(* IEC 61131-3 sources: SmartHomeNew/snapshots/2026-05-19, 186 files *)

(* ---- E_Adapt_Profile.dut ---- *)
{attribute 'strict'}
TYPE E_Adapt_Profile :
(
    ADAPT_PROFILE_STABLE := 0,
    ADAPT_PROFILE_BALANCED := 1,
    ADAPT_PROFILE_AGGRESSIVE := 2
) USINT;
END_TYPE

(* ---- E_FABRIC_LIFECYCLE_STATE.dut ---- *)
TYPE E_FABRIC_LIFECYCLE_STATE : (
    FABRIC_INITIALIZING,
    FABRIC_ACTIVE,
    FABRIC_DEGRADED,
    FABRIC_PASSIVE,
    FABRIC_QUARANTINED,
    FABRIC_SUSPENDED
);
END_TYPE

(* ---- E_GOVERNANCE_PRIORITY_TIER.dut ---- *)
TYPE E_GOVERNANCE_PRIORITY_TIER : (
    TIER_0_SAFETY,
    TIER_1_AUTHORITY,
    TIER_2_PHYSICAL_TRUTH,
    TIER_3_SURVIVABILITY,
    TIER_4_OBSERVABILITY,
    TIER_5_ANALYTICS
);
END_TYPE

(* ---- E_Heating_Allocation_Block_Reason.dut ---- *)
TYPE E_Heating_Allocation_Block_Reason :
(
    NONE := 0,
    PRESSURE_UNAVAILABLE := 1,
    SERVICE_DISABLED := 2,
    PREDICTIVE_DEGRADED := 3,
    POLICY_BUDGET_SHED := 4,
    FREEZE_BYPASS := 5,
    DHW_BYPASS := 6
);
END_TYPE

(* ---- E_OpenTherm_Adapter_State.dut ---- *)
TYPE E_OpenTherm_Adapter_State :
(
    OT_STATE_OFFLINE := 0,
    OT_STATE_ONLINE := 1,
    OT_STATE_HEARTBEAT_TIMEOUT := 2,
    OT_STATE_ACK_TIMEOUT := 3,
    OT_STATE_ADAPTER_ERROR := 4
);
END_TYPE

(* ---- E_PLC_ROLE.dut ---- *)
{attribute 'strict'}
TYPE E_PLC_ROLE :
(
    ROLE_UNDEFINED := 0,
    ROLE_ACTIVE := 1,
    ROLE_STANDBY := 2,
    ROLE_OFFLINE := 3
) USINT;
END_TYPE

(* ---- E_Runtime_Observer_Lifecycle_State.dut ---- *)
TYPE E_Runtime_Observer_Lifecycle_State :
(
    ROS_INACTIVE := 0,
    ROS_AUTHORIZATION_PENDING := 10,
    ROS_AUTHORIZATION_DENIED := 20,
    ROS_STABILIZATION := 30,
    ROS_OPERATIONAL := 40,
    ROS_ROLLBACK := 50,
    ROS_FAULTED := 900
);
END_TYPE

(* ---- E_SEMANTIC_EXECUTION_PATH.dut ---- *)
TYPE E_SEMANTIC_EXECUTION_PATH : (
    FAST_PATH,
    NORMAL_PATH,
    DEFERRED_PATH,
    BACKGROUND_PATH
);
END_TYPE

(* ---- E_System_Reason_Code.dut ---- *)
{attribute 'strict'}
TYPE E_System_Reason_Code :
(
    REASON_NONE := 0,
    REASON_USER := 1,
    REASON_SAFETY := 2,
    REASON_AUTOMATION := 3,
    REASON_INTERNAL := 4,
    REASON_SCENARIO_VENT_BOOST := 5,
    REASON_USER_REQUEST := 6,
    REASON_SCENARIO_NIGHT := 7,
    REASON_DOMAIN_PROJECTION := 8,
    REASON_SAFETY_BLOCK := 9
) USINT;
END_TYPE

(* ---- E_SYSTEM_RUNTIME_STATE.dut ---- *)
TYPE E_SYSTEM_RUNTIME_STATE : (
    SYS_SAFE,
    SYS_DEGRADED,
    SYS_RECOVERING,
    SYS_QUARANTINED,
    SYS_ISOLATED,
    SYS_PARTITIONED,
    SYS_TRUSTLESS
);
END_TYPE

(* ---- E_VALVE_TYPE.dut ---- *)
{attribute 'strict'}
TYPE E_VALVE_TYPE :
(
  VALVE_NC := 1,
  VALVE_NO := 2
) USINT;
END_TYPE

(* ---- E_WEATHER_COMPENSATION_METHOD.dut ---- *)
{attribute 'strict'}
TYPE E_WEATHER_COMPENSATION_METHOD :
(
  WEATHER_COMP_NONE := 0,
  WEATHER_COMP_OUTDOOR_RESET := 1
) USINT;
END_TYPE

(* ---- GVL_FABRIC_LIFECYCLE_REGISTRY.gvl ---- *)
TYPE E_FABRIC_LIFECYCLE_STATE : (
    FABRIC_INITIALIZING,
    FABRIC_ACTIVE,
    FABRIC_DEGRADED,
    FABRIC_PASSIVE,
    FABRIC_QUARANTINED,
    FABRIC_SUSPENDED
);
END_TYPE

TYPE E_RUNTIME_ADAPTIVE_MODE : (
    FULL_SEMANTIC_MODE,
    REDUCED_ANALYTICS_MODE,
    SURVIVABILITY_MODE,
    MINIMAL_SAFE_MODE
);
END_TYPE

VAR_GLOBAL
    // Lifecycle governance.
    Fabric_Lifecycle_Registry_Active : BOOL := TRUE;
    Fabric_Lifecycle_Registry_ReadOnly : BOOL := TRUE;

    Runtime_Adaptive_Mode : E_RUNTIME_ADAPTIVE_MODE := FULL_SEMANTIC_MODE;

    // Major fabric lifecycle states.
    Safety_Fabric_State : E_FABRIC_LIFECYCLE_STATE := FABRIC_ACTIVE;
    Authority_Fabric_State : E_FABRIC_LIFECYCLE_STATE := FABRIC_ACTIVE;
    Physical_Reality_Fabric_State : E_FABRIC_LIFECYCLE_STATE := FABRIC_ACTIVE;
    Survivability_Fabric_State : E_FABRIC_LIFECYCLE_STATE := FABRIC_ACTIVE;
    Observability_Fabric_State : E_FABRIC_LIFECYCLE_STATE := FABRIC_ACTIVE;
    Analytics_Fabric_State : E_FABRIC_LIFECYCLE_STATE := FABRIC_ACTIVE;

    // Controlled capability shedding advisories.
    Controlled_Capability_Shedding_Allowed : BOOL := FALSE;
    NonEssential_Analytics_Shedding_Recommended : BOOL := FALSE;
    Extended_Observability_Shedding_Recommended : BOOL := FALSE;
    Simulation_Suspension_Recommended : BOOL := FALSE;
    Diagnostics_Degradation_Recommended : BOOL := FALSE;

    // Critical fabrics never shed.
    Safety_Fabric_Protected : BOOL := TRUE;
    Authority_Fabric_Protected : BOOL := TRUE;
    Physical_Reality_Fabric_Protected : BOOL := TRUE;
    Runtime_Barrier_Protected : BOOL := TRUE;

    // Recovery-aware restoration.
    Gradual_Reactivation_Allowed : BOOL := FALSE;
    Stability_Validated_Reactivation_Required : BOOL := TRUE;

    Fabric_Lifecycle_Registry_Epoch : UDINT := 0;
END_VAR

(* ---- GVL_RUNTIME_STATE_ALGEBRA.gvl ---- *)
TYPE E_SYSTEM_RUNTIME_STATE : (
    SYS_SAFE,
    SYS_DEGRADED,
    SYS_RECOVERING,
    SYS_QUARANTINED,
    SYS_ISOLATED,
    SYS_PARTITIONED,
    SYS_TRUSTLESS
);
END_TYPE

VAR_GLOBAL
    Current_Runtime_State : E_SYSTEM_RUNTIME_STATE := SYS_SAFE;
    Previous_Runtime_State : E_SYSTEM_RUNTIME_STATE := SYS_SAFE;

    Runtime_State_Transition_Valid : BOOL := FALSE;
    Runtime_State_Lineage_Coherent : BOOL := FALSE;
    Runtime_State_Monotonic : BOOL := FALSE;

    Runtime_State_ReadOnly_Projection : BOOL := TRUE;
    Runtime_State_NoExecutionMutation : BOOL := TRUE;

    Runtime_State_Transition_Observed : BOOL := FALSE;
    Runtime_State_Drift_Observed : BOOL := FALSE;

    Runtime_State_Epoch : UDINT := 0;
END_VAR

(* ---- GVL_RUNTIME_TRANSITION_SYSTEM.gvl ---- *)
TYPE E_RUNTIME_TRANSITION_RESULT : (
    TRANSITION_VALID,
    TRANSITION_FORBIDDEN,
    TRANSITION_REQUIRES_PROOF,
    TRANSITION_REQUIRES_RECOVERY,
    TRANSITION_REQUIRES_TEMPORAL_ALIGNMENT
);
END_TYPE

VAR_GLOBAL
    Current_Transition_Result : E_RUNTIME_TRANSITION_RESULT := TRANSITION_VALID;

    Runtime_Transition_Validation_Active : BOOL := TRUE;
    Runtime_Transition_ReadOnly_Mode : BOOL := TRUE;
    Runtime_Transition_NoMutation : BOOL := TRUE;

    Runtime_Transition_Legal : BOOL := FALSE;
    Runtime_Transition_Proofs_Valid : BOOL := FALSE;
    Runtime_Transition_Lineage_Valid : BOOL := FALSE;
    Runtime_Transition_Temporal_Valid : BOOL := FALSE;

    Illegal_Runtime_Transition_Observed : BOOL := FALSE;
    Unsafe_State_Promotion_Observed : BOOL := FALSE;
    Recovery_Without_Lineage_Observed : BOOL := FALSE;
    Unsafe_Trust_Escalation_Observed : BOOL := FALSE;

    Runtime_Transition_Epoch : UDINT := 0;
END_VAR

(* ---- GVL_TRACE.gvl ---- *)
TYPE E_Trace_Layer :
(
    TRACE_SENSOR,
    TRACE_SCENARIO,
    TRACE_INTENT,
    TRACE_COMMAND,
    TRACE_DOMAIN,
    TRACE_IO,
    TRACE_SAFETY,
    TRACE_RECOVERY,
    TRACE_USER
);
END_TYPE

TYPE E_Trace_Source :
(
    SRC_NONE,
    SRC_SENSOR,
    SRC_USER,
    SRC_SCENARIO,
    SRC_SAFETY,
    SRC_RECOVERY,
    SRC_COMMAND,
    SRC_DOMAIN,
    SRC_IO
);
END_TYPE

TYPE ST_Trace_Entry :
STRUCT
    Timestamp_MS : UDINT;
    Layer : E_Trace_Layer;
    Source : E_Trace_Source;
    Reason_Code : E_System_Reason_Code;
    Value_Bool : BOOL;
    Value_Real : REAL;
    Text : STRING(120);
END_STRUCT
END_TYPE

VAR_GLOBAL
    G_Trace_Buffer : ARRAY[1..200] OF ST_Trace_Entry;
    G_Trace_Write_Index : INT := 1;
    G_Trace_Enabled : BOOL := TRUE;
END_VAR

(* ---- ST_DHW_Config.dut ---- *)
{attribute 'pack_mode' := '1'}
TYPE ST_DHW_Config :
STRUCT
    Target_Temp : REAL := 55.0;
    Hysteresis : REAL := 2.0;
    Circulation_Schedule_Enabled : BOOL := TRUE;
    Circulation_Start : TOD := TOD#06:00;
    Circulation_End : TOD := TOD#23:00;
    Night_Mode_Enabled : BOOL := TRUE;
    Anti_Legionella_Enabled : BOOL := TRUE;
    Anti_Legionella_Day : UINT := 7;
    Degraded_Target_Delta : REAL := 5.0; // Снижение целевой температуры ГВС в режиме DEGRADED
END_STRUCT
END_TYPE

(* ---- ST_Distributed_Recovery_Lock.dut ---- *)
TYPE ST_Distributed_Recovery_Lock :
STRUCT
    Lock_Valid : BOOL;
    Runtime_System_Time_MS : UDINT;

    Lock_Id : UDINT;
    Lock_Sequence_Id : UDINT;

    Owner_Controller_Id : UINT;
    Owner_Runtime_Node_Id : UINT;

    Recovery_Lock_Active : BOOL;
    Rollback_Lock_Active : BOOL;
    Reopen_Lock_Active : BOOL;

    Lock_Conflict : BOOL;
    Lock_Expired : BOOL;
    Lock_Revoked : BOOL;

    Distributed_Execution_Allowed : BOOL;

    Status_Code : UINT;
    Status_Text : STRING(160);
END_STRUCT
END_TYPE

(* ---- ST_Distributed_Runtime_Message.dut ---- *)
TYPE ST_Distributed_Runtime_Message :
STRUCT
    Message_Valid : BOOL;
    Message_Time_MS : UDINT;
    Message_Id : UDINT;

    Source_Controller_Id : UINT;
    Source_Runtime_Node_Id : UINT;
    Target_Runtime_Node_Id : UINT;

    Message_Class : UINT;
    Message_Version : UINT;

    Authority_State_Replicated : BOOL;
    Recovery_State_Replicated : BOOL;
    Quarantine_State_Replicated : BOOL;
    Topology_State_Replicated : BOOL;
    Binding_State_Replicated : BOOL;

    Replication_Sequence_Id : UDINT;
    Replication_Ack_Required : BOOL;
    Replication_Ack_Received : BOOL;

    Status_Code : UINT;
    Status_Text : STRING(160);
END_STRUCT
END_TYPE

(* ---- ST_FloorHeating_Global_Config.dut ---- *)
{attribute 'pack_mode' := '1'}
TYPE ST_FloorHeating_Global_Config :
STRUCT
    enable_floor_heating : BOOL := TRUE;
    anti_freeze_temp : REAL := 7.0;
    overheat_temp : REAL := 45.0;
    weather_compensation_enabled : BOOL := TRUE;
    total_circuits : BYTE := 16;
END_STRUCT
END_TYPE

(* ---- ST_FloorHeating_Manifold_Config.dut ---- *)
{attribute 'pack_mode' := '1'}
TYPE ST_FloorHeating_Manifold_Config :
STRUCT
    manifold_id : BYTE;
    location : STRING(30);
    nominal_flow : REAL;
    enable_pump : BOOL;
    circuits : ARRAY[1..GVL_CONSTANTS.C_MAX_CIRCUITS_PER_MANIFOLD] OF ST_FloorHeating_Circuit_Config;
END_STRUCT
END_TYPE

(* ---- ST_Heating_Runtime_Anomaly.dut ---- *)
TYPE ST_Heating_Runtime_Anomaly :
STRUCT
    // ======================================================
    // Anomaly lifecycle
    // ======================================================
    Anomaly_Active : BOOL;
    Anomaly_Acknowledged : BOOL;
    Anomaly_Cleared : BOOL;

    // ======================================================
    // Runtime anomaly sources
    // ======================================================
    Runtime_Jitter_Detected : BOOL;
    Runtime_Latency_Detected : BOOL;
    Runtime_Degraded : BOOL;

    // ======================================================
    // Cascade anomaly sources
    // ======================================================
    Cascade_Degraded : BOOL;
    Cascade_Boiler_Loss_Detected : BOOL;

    // ======================================================
    // OpenTherm anomaly sources
    // ======================================================
    OpenTherm_Transport_Degraded : BOOL;
    OpenTherm_Command_Invalid : BOOL;

    // ======================================================
    // Diagnostics anomaly sources
    // ======================================================
    Diagnostics_Degraded : BOOL;
    Explainability_Degraded : BOOL;

    // ======================================================
    // Runtime integrity
    // ======================================================
    Sequencing_Invalid : BOOL;
    Ownership_Invalid : BOOL;
    Synchronization_Invalid : BOOL;

    // ======================================================
    // Anomaly severity
    // ======================================================
    Severity_Level : UINT;
    Critical_Anomaly : BOOL;

    // ======================================================
    // Runtime status
    // ======================================================
    Status_Code : UINT;
    Status_Text : STRING(128);
END_STRUCT
END_TYPE

(* ---- ST_Heating_Runtime_Blackbox_Event.dut ---- *)
TYPE ST_Heating_Runtime_Blackbox_Event :
STRUCT
    // ======================================================
    // Event identity
    // ======================================================
    Event_ID : UDINT;
    Event_Active : BOOL;

    // ======================================================
    // Runtime phase
    // ======================================================
    Runtime_Phase : E_Heating_Runtime_Phase;

    // ======================================================
    // Event timing
    // ======================================================
    Event_Start_MS : UDINT;
    Event_End_MS : UDINT;
    Event_Duration_MS : UDINT;

    // ======================================================
    // Runtime degradation state
    // ======================================================
    Runtime_Degraded : BOOL;
    Runtime_Fault : BOOL;

    // ======================================================
    // Cascade state
    // ======================================================
    Cascade_Degraded : BOOL;
    Cascade_Boiler_Loss : BOOL;

    // ======================================================
    // OpenTherm state
    // ======================================================
    OpenTherm_Degraded : BOOL;
    OpenTherm_Command_Invalid : BOOL;

    // ======================================================
    // Integrity state
    // ======================================================
    Sequencing_Invalid : BOOL;
    Ownership_Invalid : BOOL;
    Synchronization_Invalid : BOOL;

    // ======================================================
    // Root-cause state
    // ======================================================
    Root_Cause_Candidate : BOOL;
    Critical_Path : BOOL;

    // ======================================================
    // Event status
    // ======================================================
    Status_Code : UINT;
    Status_Text : STRING(128);
END_STRUCT
END_TYPE

(* ---- ST_Heating_Runtime_Causality_Graph.dut ---- *)
TYPE ST_Heating_Runtime_Causality_Graph :
STRUCT
    // ======================================================
    // Graph nodes
    // ======================================================
    Nodes : ARRAY[1..64] OF ST_Heating_Runtime_Causality_Node;

    // ======================================================
    // Graph edges
    // ======================================================
    Edges : ARRAY[1..128] OF ST_Heating_Runtime_Causality_Edge;

    // ======================================================
    // Graph state
    // ======================================================
    Node_Count : UINT;
    Edge_Count : UINT;

    Graph_Active : BOOL;
    Graph_Degraded : BOOL;
    Graph_Critical : BOOL;

    // ======================================================
    // Graph integrity
    // ======================================================
    Sequencing_Valid : BOOL;
    Ownership_Valid : BOOL;
    Synchronization_Valid : BOOL;

    // ======================================================
    // Graph status
    // ======================================================
    Status_Code : UINT;
    Status_Text : STRING(128);
END_STRUCT
END_TYPE

(* ---- ST_Heating_Runtime_Execution_Timeline.dut ---- *)
TYPE ST_Heating_Runtime_Execution_Timeline :
STRUCT
    // ======================================================
    // Execution frames
    // ======================================================
    Frames : ARRAY[1..64] OF ST_Heating_Runtime_Execution_Frame;

    // ======================================================
    // Timeline state
    // ======================================================
    Write_Index : UINT;
    Frame_Count : UINT;
    Timeline_Overflow : BOOL;

    // ======================================================
    // Timeline integrity
    // ======================================================
    Sequencing_Valid : BOOL;
    Ownership_Valid : BOOL;
    Synchronization_Valid : BOOL;

    // ======================================================
    // Timeline telemetry
    // ======================================================
    Runtime_Jitter_Detected : BOOL;
    Runtime_Latency_Detected : BOOL;
    Runtime_Degraded : BOOL;

    // ======================================================
    // Timeline status
    // ======================================================
    Status_Code : UINT;
    Status_Text : STRING(128);
END_STRUCT
END_TYPE

(* ---- ST_Heating_Runtime_Meta_Supervision.dut ---- *)
TYPE ST_Heating_Runtime_Meta_Supervision :
STRUCT
    // ======================================================
    // Meta-analytics visibility
    // Passive governance analytics only.
    // No supervisory authority exists.
    // ======================================================
    Meta_Analytics_Visible : BOOL;
    Meta_Analytics_Degraded : BOOL;
    Meta_Analytics_Attention : BOOL;

    // ======================================================
    // Supervision integrity observation
    // ======================================================
    Supervision_Integrity_Visible : BOOL;
    Supervision_Integrity_Observation : UINT;

    // ======================================================
    // Adaptive supervision drift observation
    // ======================================================
    Adaptive_Drift_Visible : BOOL;
    Adaptive_Drift_Observation : UINT;

    // ======================================================
    // Predictive confidence observation
    // ======================================================
    Confidence_Degradation_Visible : BOOL;
    Confidence_Degradation_Observation : UINT;

    // ======================================================
    // Analytics consistency observation
    // ======================================================
    Analytics_Consistency_Visible : BOOL;
    Analytics_Consistency_Observation : UINT;

    // ======================================================
    // Meta integrity observation
    // ======================================================
    Sequencing_Meta_Observation : BOOL;
    Ownership_Meta_Observation : BOOL;
    Synchronization_Meta_Observation : BOOL;

    // ======================================================
    // Meta-analytics status
    // ======================================================
    Status_Code : UINT;
    Status_Text : STRING(128);
END_STRUCT
END_TYPE

(* ---- ST_Input_Quality_Record.dut ---- *)
TYPE ST_Input_Quality_Record :
STRUCT
    Quality_Visible : BOOL;
    Value_Valid : BOOL;
    Value_Degraded : BOOL;
    Spike_Detected : BOOL;
    Stuck_Detected : BOOL;
    Confidence : REAL;
    Last_Value : REAL;
    Last_Change_MS : UDINT;
    Reason_Code : UINT;
    Reason_Text : STRING(128);
END_STRUCT
END_TYPE

(* ---- ST_Manifold_Status.dut ---- *)
{attribute 'pack_mode' := '1'}
TYPE ST_Manifold_Status :
STRUCT
    Pump_On : BOOL;
    Pump_Current : REAL;
    Pressure : REAL;
    Temp_Supply : REAL;
    Temp_Return : REAL;
    Valve_Pos : REAL;
    Error : BOOL;
    Error_ID : WORD;
    Health : ST_Device_Health; // Диагностика насоса
END_STRUCT
END_TYPE

(* ---- ST_Owen_Analog_Value.dut ---- *)
{attribute 'pack_mode' := '1'}
TYPE ST_Owen_Analog_Value :
STRUCT
    rValue : REAL;
    uiCycleTime : UINT;
    wStatus : WORD;
END_STRUCT
END_TYPE

(* ---- ST_Rule.dut ---- *)
TYPE ST_Rule :
STRUCT
    Action_Type : INT;
    Action_Target_ID : INT;
    Action_Value : REAL;

    Condition_Type : INT;
    Condition_Target_ID : INT;
    Condition_Op : INT;
    Condition_Value : REAL;
    Condition_Value_Max : REAL;
END_STRUCT
END_TYPE

(* ---- ST_Runtime_Bus_Frame.dut ---- *)
TYPE ST_Runtime_Bus_Frame :
STRUCT
    Frame_Valid : BOOL;
    Frame_Time_MS : UDINT;
    Frame_Id : UDINT;

    Source_Controller_Id : UINT;
    Source_Runtime_Node_Id : UINT;
    Target_Runtime_Node_Id : UINT;

    Frame_Class : UINT;
    Frame_Sequence_Id : UDINT;
    Frame_Ack_Required : BOOL;
    Frame_Ack_Received : BOOL;

    Authority_State_Frame : BOOL;
    Recovery_State_Frame : BOOL;
    Quarantine_State_Frame : BOOL;
    Topology_State_Frame : BOOL;
    Binding_State_Frame : BOOL;
    Predictive_State_Frame : BOOL;

    Replication_Consistent : BOOL;
    Replication_Stale : BOOL;
    Replication_Rejected : BOOL;

    Status_Code : UINT;
    Status_Text : STRING(160);
END_STRUCT
END_TYPE

(* ---- ST_Scenario_Stats.dut ---- *)
TYPE ST_Scenario_Stats :
STRUCT
    Activations : UDINT;
    Success_Count : UDINT;
    Failure_Count : UDINT;
    Success_Rate : REAL;
    Avg_Result_Value : REAL;
    Stability_Counter : INT;
    Last_Activation : UDINT;
END_STRUCT
END_TYPE

(* ---- ST_Security_Global_Config.dut ---- *)
{attribute 'pack_mode' := '1'}
TYPE ST_Security_Global_Config :
STRUCT
    PIN_Code : STRING(4) := '1234';
    Phones : ARRAY[1..GVL_CONSTANTS.C_MAX_SECURITY_PHONES] OF STRING(15);
    entry_delay_seconds : UDINT := 30;
    exit_delay_seconds : UDINT := 60;
    alarm_duration_seconds : UDINT := 180;
    two_person_timeout_seconds : UDINT := 120;
    max_access_attempts : BYTE := 3;
    auto_arm_enabled : BOOL := FALSE;
    auto_arm_time_ms : UDINT := 0;
    enable_2fa : BOOL := TRUE; // Включение/отключение двухфакторной аутентификации
    gate_open_pulse_ms : UDINT := GVL_CONSTANTS.C_MS_IN_SECOND;
    wicket_open_pulse_ms : UDINT := GVL_CONSTANTS.C_MS_IN_SECOND;
    lock_open_pulse_ms : UDINT := GVL_CONSTANTS.C_MS_IN_SECOND;
    lock_close_pulse_ms : UDINT := GVL_CONSTANTS.C_MS_IN_SECOND;

    // Байпасы зон
    bypass_motion : ARRAY[1..16] OF BOOL;
    bypass_doors : ARRAY[1..GVL_CONSTANTS.C_MAX_DOOR_SENSORS] OF BOOL;
    bypass_windows : ARRAY[1..16] OF BOOL;
END_STRUCT
END_TYPE

(* ---- ST_Security_Zone_State.dut ---- *)
{attribute 'pack_mode' := '1'}
TYPE ST_Security_Zone_State :
STRUCT
    Armed : BOOL;
    Alarm : BOOL;
    Bypassed : BOOL;
    Last_Trigger_Time : DT;
    Trigger_Count : UINT;
END_STRUCT
END_TYPE

(* ---- ST_Sensor_Calibration_Record.dut ---- *)
{attribute 'pack_mode' := '1'}
TYPE ST_Sensor_Calibration_Record :
STRUCT
    sensor_id : UDINT := 0;
    sensor_type : E_SENSOR_TYPE;
    zone_id : BYTE := 0;
    offset : REAL := 0.0;
    multiplier : REAL := 1.0;
    last_calibration_timestamp : UDINT := 0;
    verification_passed : BOOL := FALSE;
END_STRUCT
END_TYPE

(* ---- ST_Trend_Header.dut ---- *)
{attribute 'pack_mode' := '1'}
TYPE ST_Trend_Header :
STRUCT
    parameter_type : BYTE; // E_Trend_Parameter_Type
    zone_id : BYTE := 0;
    records_count : UDINT := 0;
    average_value : REAL := 0.0;
    min_value : REAL := 0.0;
    max_value : REAL := 0.0;
END_STRUCT
END_TYPE

(* ---- ST_TwoFactor_Auth_State.dut ---- *)
TYPE ST_TwoFactor_Auth_State :
STRUCT
    Auth_Method : E_TwoFactor_Method;
    is_pending : BOOL;
    Attempts_Left : UINT;
    Time_Left_S : UINT;
    Is_Success : BOOL;
    Is_Locked : BOOL;
END_STRUCT
END_TYPE

(* ---- ST_Ventilation_Unit.dut ---- *)
{attribute 'pack_mode' := '1'}
TYPE ST_Ventilation_Unit :
STRUCT
    Enabled : BOOL;
    Speed_Percent : REAL;
    Filter_Dirty : BOOL;
    Error : BOOL;
    Mode : BYTE;
END_STRUCT
END_TYPE

(* ---- ST_Water_Event_Log_Record.dut ---- *)
TYPE ST_Water_Event_Log_Record : STRUCT Runtime_Valid : BOOL; Event_Time_MS : UDINT; Event_Id : UINT; Event_Text : STRING(80); END_STRUCT END_TYPE

(* ---- ST_Water_Hydraulic_Topology_Edge.dut ---- *)
TYPE ST_Water_Hydraulic_Topology_Edge :
STRUCT
    Runtime_Valid : BOOL;

    Edge_Id : UINT;

    Upstream_Segment_Id : UINT;
    Downstream_Segment_Id : UINT;

    Isolation_Group_Id : UINT;
    Valve_Group_Id : UINT;

    Shared_Trunk : BOOL;
    Cross_Zone_Dependency : BOOL;

    Dependency_Valid : BOOL;
    Dependency_Ambiguous : BOOL;

    Selective_Isolation_Allowed : BOOL;
    Global_Fallback_Required : BOOL;

    Status_Code : UINT;
    Status_Text : STRING(128);
END_STRUCT
END_TYPE

(* ---- ST_Water_Output_Reconciliation_State.dut ---- *)
TYPE ST_Water_Output_Reconciliation_State :
STRUCT
    Runtime_Valid : BOOL;
    Runtime_System_Time_MS : UDINT;

    Valve_Group_Id : UINT;

    Projection_Active : BOOL;
    Runtime_Output_Active : BOOL;

    Expected_Closed : BOOL;
    Confirmed_Closed : BOOL;
    Confirmation_Unknown : BOOL;

    Reconciliation_Healthy : BOOL;
    Projection_Runtime_Mismatch : BOOL;
    Projection_Confirmation_Mismatch : BOOL;

    Conflict_Detected : BOOL;
    Topology_Invalid : BOOL;

    Status_Code : UINT;
    Status_Text : STRING(128);
END_STRUCT
END_TYPE

(* ---- ST_Water_Physical_Convergence_State.dut ---- *)
TYPE ST_Water_Physical_Convergence_State :
STRUCT
    Runtime_Valid : BOOL;
    Runtime_System_Time_MS : UDINT;

    Sensor_Id : UINT;

    Projection_Active : BOOL;
    Physical_State_Confirmed : BOOL;
    Runtime_Converged : BOOL;

    Physical_Open_Confirmed : BOOL;
    Physical_Closed_Confirmed : BOOL;

    Projection_Mismatch : BOOL;
    Runtime_Mismatch : BOOL;
    Physical_Mismatch : BOOL;

    Convergence_Degraded : BOOL;
    Escalation_Required : BOOL;

    Status_Code : UINT;
    Status_Text : STRING(128);
END_STRUCT
END_TYPE

(* ---- GVL_AUTHORITY_RESTORATION.gvl ---- *)
VAR_GLOBAL
    // Global authority restoration governance.
    Authority_Restoration_Active : BOOL := FALSE;
    Authority_Restoration_Allowed : BOOL := FALSE;
    Authority_Restoration_Completed : BOOL := FALSE;

    // Staged re-authorization.
    Snapshot_Restoration_Valid : BOOL := FALSE;
    Consensus_Restoration_Valid : BOOL := FALSE;
    Causality_Restoration_Valid : BOOL := FALSE;
    Epoch_Restoration_Valid : BOOL := FALSE;
    Lineage_Restoration_Valid : BOOL := FALSE;

    // Quarantine exit ordering.
    Revocation_Clearance_Valid : BOOL := FALSE;
    Stabilization_Window_Elapsed : BOOL := FALSE;
    Reauthorization_Order_Valid : BOOL := FALSE;

    // Restoration protection.
    Premature_Restoration_Detected : BOOL := FALSE;
    Partial_Restoration_Detected : BOOL := FALSE;
    Restoration_Replay_Suspected : BOOL := FALSE;
    Quarantine_Exit_Race_Detected : BOOL := FALSE;

    // Temporal authority.
    Restoration_Epoch : UDINT := 0;
    Restoration_Last_Update_MS : UDINT := 0;

    // Diagnostics.
    Restoration_Last_Error_Code : UDINT := 0;
    Restoration_Last_Error_Text : STRING(160) := '';
    Restoration_Invalidation_Count : UDINT := 0;
END_VAR

(* ---- GVL_AUTHORITY_REVOCATION.gvl ---- *)
VAR_GLOBAL
    // Global revocation authority.
    Authority_Revocation_Active : BOOL := FALSE;
    Authority_Revocation_Propagated : BOOL := FALSE;
    Authority_Fail_Closed_Valid : BOOL := FALSE;

    // Upstream invalidation sources.
    Snapshot_Authority_Revoked : BOOL := FALSE;
    Sensor_Consensus_Authority_Revoked : BOOL := FALSE;
    Telemetry_Causality_Authority_Revoked : BOOL := FALSE;
    Physical_Authority_Epoch_Revoked : BOOL := FALSE;
    Authority_Lineage_Revoked : BOOL := FALSE;

    // Downstream revocation guarantees.
    PreOutput_Authority_Revoked : BOOL := FALSE;
    Physical_IO_Release_Denied : BOOL := FALSE;
    Quarantine_Fabric_Active : BOOL := FALSE;

    // Ordering/coherence protection.
    Revocation_Order_Valid : BOOL := FALSE;
    Revocation_Replay_Suspected : BOOL := FALSE;
    Partial_Revocation_Detected : BOOL := FALSE;
    Stale_Downstream_Authority_Detected : BOOL := FALSE;

    // Temporal authority.
    Revocation_Epoch : UDINT := 0;
    Revocation_Last_Update_MS : UDINT := 0;

    // Diagnostics.
    Revocation_Last_Error_Code : UDINT := 0;
    Revocation_Last_Error_Text : STRING(160) := '';
    Revocation_Invalidation_Count : UDINT := 0;
END_VAR

(* ---- GVL_COMMAND.gvl ---- *)
{attribute 'qualified_only'}
VAR_GLOBAL
    // ======================================================
    // LEGACY / OPERATOR COMMAND REQUEST SURFACE
    // ======================================================
    // This GVL is retained as legacy/operator command request
    // surface and comparison source for command verification.
    //
    // Runtime operational command ownership lives in
    // GVL_COMMAND_SHADOW and is published by PRG_Command_Arbitration.
    //
    // PreOutput and Command_Verifier may compare this surface against
    // GVL_COMMAND_SHADOW, but must not treat GVL_COMMAND as final
    // physical output authority.
    // ======================================================

    G_Gas_Valve_Close : BOOL := FALSE;
    G_Boiler_Stop : BOOL := FALSE;
    G_Supply_100_Req : BOOL := FALSE;
    G_Supply_80_Req : BOOL := FALSE;
    G_Vent_PV3_Boost : BOOL := FALSE;
    G_Exhaust_100_Req : BOOL := FALSE;
    G_Vent_Stop : BOOL := FALSE;
    G_Close_Valve_35 : BOOL := FALSE;
    G_Close_Valve_36 : BOOL := FALSE;
    G_Gate_Open : BOOL;
    G_Wicket_Open : BOOL;
    G_Lock_1_Open : BOOL;
    G_Lock_1_Close : BOOL;
    G_Lock_2_Open : BOOL;
    G_Lock_2_Close : BOOL;
    G_Reset_Errors : BOOL := FALSE;
    G_Scenario_Request : E_SCENARIO_TYPE := E_SCENARIO_TYPE.SCENARIO_NONE;
    G_Scenario_Request_Operator : E_SCENARIO_TYPE := E_SCENARIO_TYPE.SCENARIO_NONE;

    G_Arm_Req : BOOL;
    G_Disarm_Req : BOOL;
    G_PIN_Code : STRING(4);
    G_RFID_Tag : STRING(20);
    G_2FA_Code_In : STRING(6);
    G_Send_2FA_Req : BOOL;
    G_2FA_Code_Out : STRING(6);
    G_Lighting_Override : ARRAY[1..GVL_CONSTANTS.C_MAX_LIGHT_ZONES] OF BYTE;
    G_Blinds_Override : ARRAY[1..GVL_CONSTANTS.C_MAX_BLINDS] OF BYTE;
    G_Socket_Override : ARRAY[1..GVL_CONSTANTS.C_MAX_SOCKETS] OF BOOL;
    CMD_Set_Manifold_Pump_In_Service : ARRAY[1..GVL_CONSTANTS.C_MAX_MANIFOLDS] OF BOOL;
    CMD_Set_DHW_Heating_Pump_In_Service : BOOL;
    CMD_Set_DHW_Circ_Pump_In_Service : BOOL;
    CMD_Dangerous_Action_Confirm : BOOL;
    CMD_Dangerous_Action_Request : BOOL;
    CMD_User_Access_Level : INT := 0;
    CMD_Valve_Test_Open : BOOL;
    CMD_Valve_Test_Close : BOOL;
    CMD_Valve_Test_Confirm : BOOL;
    CMD_Water_Valve_Test_Open : BOOL;
    CMD_Water_Valve_Test_Close : BOOL;
    CMD_Water_Valve_Test_Confirm : BOOL;
    CMD_Gas_Valve_Test_Open : BOOL;
    CMD_Gas_Valve_Test_Close : BOOL;
    CMD_Gas_Valve_Test_Confirm : BOOL;
    CMD_Water_Selective_Recover : BOOL;
    CMD_Gas_Selective_Recover : BOOL;
END_VAR

(* ---- GVL_COMMAND_SHADOW.gvl ---- *)
VAR_GLOBAL
    // ======================================================
    // OPERATIONAL COMMAND SHADOW STATE
    // ======================================================
    // Operational command layer produced exclusively by
    // PRG_Command_Arbitration during migration.
    //
    // Downstream execution layers consume these fields as read-only.
    // PreOutput barriers, verifier layers and IO publication layers
    // must not mutate command shadow ownership state.
    // ======================================================

    // Gas / boiler / ventilation
    G_Gas_Valve_Close : BOOL := FALSE;
    G_Boiler_Stop : BOOL := FALSE;
    G_Supply_100_Req : BOOL := FALSE;
    G_Supply_80_Req : BOOL := FALSE;
    G_Vent_PV3_Boost : BOOL := FALSE;
    G_Exhaust_100_Req : BOOL := FALSE;
    G_Vent_Stop : BOOL := FALSE;
    G_Vent_Block : BOOL := FALSE;
    G_Vent_Smoke_Exhaust : BOOL := FALSE;

    // Heating domain command gates
    G_Heating_Block : BOOL := FALSE;
    G_Heating_Emergency_Stop : BOOL := FALSE;
    G_Heating_Gas_Safety_Stop : BOOL := FALSE;

    // Water domain command gates
    G_Water_Block : BOOL := FALSE;
    G_Water_Emergency_Stop : BOOL := FALSE;
    G_Close_Valve_35 : BOOL := FALSE;
    G_Close_Valve_36 : BOOL := FALSE;

    // Access / evacuation locks
    G_Lock_1_Open : BOOL := FALSE;
    G_Lock_1_Close : BOOL := FALSE;
    G_Lock_2_Open : BOOL := FALSE;
    G_Lock_2_Close : BOOL := FALSE;
    G_Gate_Open : BOOL := FALSE;
    G_Wicket_Open : BOOL := FALSE;
END_VAR

(* ---- GVL_CONFIG.gvl ---- *)
{attribute 'qualified_only'}
VAR_GLOBAL
    // Subsystem Configurations
    G_Heating_Config : ST_Heating_Config;
    G_DHW_Config : ST_DHW_Config;
    G_Security_Config : ST_Security_Global_Config;

    // HMI Configurations
    G_HMI_FloorHeating_Configs : ARRAY[1..GVL_CONSTANTS.C_MAX_HEATING_CIRCUITS] OF ST_FloorHeating_Circuit_Config;
    G_Heating_Circuit_To_Zone : ARRAY[1..GVL_CONSTANTS.C_MAX_HEATING_CIRCUITS] OF INT := [1, 2, 3, 4, 5, 6, 7, 8, 9, 10, 11, 12, 13, 14, 15, 16];
    G_Wet_Zone_Map : ARRAY[1..32] OF BOOL;
    G_HMI_Tariff_Settings : ST_Tariff_Config;
    G_HMI_Vent_Global_Config : ST_Ventilation_Global_Config;
    G_HMI_Scenario_Configs : ARRAY[1..GVL_CONSTANTS.C_MAX_SCENARIOS] OF ST_Scenario_Config;
    G_HMI_Flood_Config : ST_Flood_Global_Config;
    G_Flood_Global_Config : ST_Flood_Global_Config;
    G_HMI_User_Rules : ARRAY[1..GVL_CONSTANTS.C_MAX_RULES] OF ST_User_Rule;

    // Sensor calibration pipeline
    G_Calib_Outdoor_Temp : ST_Sensor_Calibration_Record;
    G_Calib_Supply_Temps : ARRAY[1..GVL_CONSTANTS.C_MAX_SUPPLY_TEMPS] OF ST_Sensor_Calibration_Record;
    G_Calib_Room_Temps : ARRAY[1..GVL_CONSTANTS.C_MAX_ZONES] OF ST_Sensor_Calibration_Record;
    G_Calib_Floor_Temps : ARRAY[1..GVL_CONSTANTS.C_MAX_ZONES] OF ST_Sensor_Calibration_Record;
    G_Calib_CO2 : ARRAY[1..GVL_CONSTANTS.C_MAX_ZONES] OF ST_Sensor_Calibration_Record;
    G_Calib_Humidity : ARRAY[1..GVL_CONSTANTS.C_MAX_ZONES] OF ST_Sensor_Calibration_Record;
    G_Calib_Manifold_T_Supply : ARRAY[1..GVL_CONSTANTS.C_MAX_MANIFOLDS] OF ST_Sensor_Calibration_Record;
    G_Calib_Manifold_T_Return : ARRAY[1..GVL_CONSTANTS.C_MAX_MANIFOLDS] OF ST_Sensor_Calibration_Record;
    G_Calib_Methane : ARRAY[1..GVL_CONSTANTS.C_MAX_METHANE_SENSORS] OF ST_Sensor_Calibration_Record;
    G_Calib_CO : ARRAY[1..GVL_CONSTANTS.C_MAX_CO_SENSORS] OF ST_Sensor_Calibration_Record;

    // Valve test configuration
    G_Valve_Test_Config : ARRAY[1..GVL_CONSTANTS.C_MAX_MANIFOLDS] OF ST_Valve_Test_Config;

    // HMI Commands & States
    G_HMI_Apply_Settings : BOOL;
    G_HMI_Mute_Alarm : BOOL;
    G_HMI_Ack_Alarms : BOOL;

    // Access Control Commands
    G_HMI_Gate_Open_Req : BOOL;
    G_HMI_Wicket_Open_Req : BOOL;
    G_HMI_Lock_1_Open_Req : BOOL;
    G_HMI_Lock_1_Close_Req : BOOL;
    G_HMI_Lock_2_Open_Req : BOOL;
    G_HMI_Lock_2_Close_Req : BOOL;
    G_Access_Pulse_MS : UDINT := 500;

    // Network security
    G_Allowed_IPs : ARRAY[1..GVL_CONSTANTS.C_MAX_ALLOWED_IPS] OF STRING(15) := ['192.168.1.100','192.168.1.101','127.0.0.1','',''];

    G_Backup_Circulation_Pump_In_Service : BOOL := TRUE;
    G_Electric_Heater_In_Service : BOOL := TRUE;
    G_Freeze_Hardware_Retry_Count : INT := 2;
    G_Freeze_Hardware_Retry_Delay_MS : UDINT := 5000;
    G_Pump_Exercise_Enabled : BOOL := TRUE;
    G_Pump_Exercise_Interval_MS : UDINT := 604800000;
    G_Pump_Exercise_Duration_MS : UDINT := 30000;
    G_Manifold_Pump_In_Service : ARRAY[1..GVL_CONSTANTS.C_MAX_MANIFOLDS] OF BOOL := [TRUE, TRUE, TRUE, TRUE, TRUE];
    G_Manifold_Priority : ARRAY[1..GVL_CONSTANTS.C_MAX_MANIFOLDS] OF INT := [3, 3, 2, 2, 1];
    G_Manifold_Thermal_Weight : ARRAY[1..GVL_CONSTANTS.C_MAX_MANIFOLDS] OF REAL := [1.0, 1.0, 0.8, 0.8, 0.5];
    G_Max_Active_Manifolds : INT := 3;
    G_Max_Thermal_Budget : REAL := 6.0;
    G_Policy_Min_Hold_MS : UDINT := 300000;
    G_DHW_Heating_Pump_In_Service : BOOL := TRUE;
    G_DHW_Circ_Pump_In_Service : BOOL := TRUE;
    G_Water_Valve_Exercise_Enabled : BOOL := TRUE;
    G_Water_Valve_Exercise_Interval_MS : UDINT := 604800000;
    G_Water_Valve_Exercise_Duration_MS : UDINT := 15000;
    G_Water_Valve_Close_Retry_Count : INT := 2;
    G_Water_Valve_Close_Retry_Delay_MS : UDINT := 3000;

    // OpenTherm / Modbus adapter configuration
    G_OpenTherm_Enabled : BOOL := FALSE;
    G_OpenTherm_Heartbeat_Timeout_MS : UDINT := 5000;
    G_OpenTherm_Command_Ack_Timeout_MS : UDINT := 3000;
    G_OpenTherm_Register_Map : ARRAY[1..GVL_CONSTANTS.C_MAX_BOILERS] OF ST_OpenTherm_Register_Map;

    // Modbus RTU transport configuration
    // Scalar fields are used instead of nested structure for CODESYS/build-system compatibility.
    G_Modbus_RTU_Driver_Attached : BOOL := FALSE;
    G_Modbus_RTU_Port_Number : BYTE := 1; // 1=COM1, 2=COM2, 3=COM3, 4=COM4
    G_Modbus_RTU_Baudrate : UDINT := 9600;
    G_Modbus_RTU_Parity : BYTE := 1; // 0=None, 1=Even, 2=Odd
    G_Modbus_RTU_Stop_Bits : BYTE := 1; // 1 or 2
    G_Modbus_RTU_Data_Bits : BYTE := 8; // usually 8
    G_Modbus_RTU_Slave_ID : BYTE := 1;
    G_Modbus_RTU_Poll_Interval_MS : UDINT := 100;
    G_Modbus_RTU_Request_Timeout_MS : UDINT := 250;
    G_Modbus_RTU_Retry_Count : INT := 2;

    // IO Mapping
    G_FloorTemp_Map : ARRAY[1..GVL_CONSTANTS.C_MAX_HEATING_CIRCUITS] OF INT := [1, 2, 3, 4, 5, 6, 7, 8, 9, 10, 11, 12, 13, 14, 15, 16];
    G_RoomTemp_Map : ARRAY[1..16] OF INT := [1, 2, 3, 4, 5, 6, 7, 8, 9, 10, 11, 12, 13, 14, 15, 16];
    G_Door_Map : ARRAY[1..GVL_CONSTANTS.C_MAX_DOOR_SENSORS] OF INT := [1, 2, 3, 4, 5, 6, 7, 8];
    G_Window_Map : ARRAY[1..16] OF INT := [9, 10, 11, 12, 13, 14, 15, 16, 17, 18, 19, 20, 21, 22, 23, 24];

    // Evacuation config
    C_MAX_LIGHT_ZONES : INT := 32;
    G_Evac_Exit_Zones : ARRAY[1..32] OF BOOL;
    G_Evac_Zone_Names : ARRAY[1..32] OF STRING(80);

END_VAR

VAR_GLOBAL CONSTANT
    C_MS_PER_SEC : UDINT := GVL_CONSTANTS.C_MS_IN_SECOND;
    C_SEC_PER_MIN : UDINT := 60;
    C_MIN_PER_HOUR : UDINT := 60;
    C_MS_PER_MIN : UDINT := GVL_CONSTANTS.C_MS_IN_MINUTE;
    C_MAX_RULES : INT := 20;
    C_ZONE_COUNT : BYTE := 18;

    ERR_PRESSURE_OUT_OF_RANGE : UDINT := 16#E004;
    ERR_HIGH_DELTA_T : UDINT := 16#E005;
    ERR_BOILER_OFFLINE : UDINT := 16#E006;
    ERR_BOILER_GENERAL_FAULT : UDINT := 16#E007;
    ERR_BOILER_NO_FLAME : UDINT := 16#E008;
    ERR_PUMP_NO_CURRENT : UDINT := 16#E009;
    ERR_PUMP_UNDERCURRENT : UDINT := 16#E00A;
    ERR_PUMP_OVERCURRENT : UDINT := 16#E00B;
    ERR_DELTA_T_LOW : UDINT := 16#E00C;
    ERR_DELTA_T_HIGH : UDINT := 16#E00D;
    ERR_DHW_IO_OFFLINE : UDINT := 16#E00E;
    ERR_DHW_TEMP_SENSOR_FAULT : UDINT := 16#E00F;
    ERR_DHW_PRESSURE_OUT_OF_RANGE : UDINT := 16#E010;
    ERR_DHW_PRESSURE_SENSOR_FAULT : UDINT := 16#E011;
    ERR_BACKUP_PUMP_OUT_OF_SERVICE : UDINT := 16#E012;
    ERR_ELECTRIC_HEATER_OUT_OF_SERVICE : UDINT := 16#E013;
    ERR_MANIFOLD_PUMP_OUT_OF_SERVICE : UDINT := 16#E014;
    ERR_DHW_HEATING_PUMP_OUT_OF_SERVICE : UDINT := 16#E015;
    ERR_DHW_CIRC_PUMP_OUT_OF_SERVICE : UDINT := 16#E016;
    ERR_FREEZE_HARDWARE_FAILED : UDINT := 16#E017;
END_VAR

(* ---- GVL_CROSSDOMAIN_FAILSAFE_CLOSURE_FABRIC.gvl ---- *)
VAR_GLOBAL
    // Deterministic cross-domain fail-safe closure governance.
    CrossDomain_FailSafe_Closure_Valid : BOOL := FALSE;
    CrossDomain_FailSafe_Closure_Granted : BOOL := FALSE;
    CrossDomain_FailSafe_Closure_Quarantine_Active : BOOL := TRUE;

    // Cross-domain fail-safe proofs.
    CrossDomain_SafeState_Compatibility_Valid : BOOL := FALSE;
    FailSafe_Topology_Closure_Canonical : BOOL := FALSE;
    MultiDomain_SafeTransition_Stable : BOOL := FALSE;
    SafeState_Recovery_Ordering_Bounded : BOOL := FALSE;
    Physical_Domain_Isolation_Coherent : BOOL := FALSE;

    // Cross-domain convergence validators.
    Thermal_Hydraulic_Compatibility_Valid : BOOL := FALSE;
    Ventilation_Heating_Compatibility_Valid : BOOL := FALSE;
    Access_Evacuation_Compatibility_Valid : BOOL := FALSE;
    Power_Recovery_Sequencing_Valid : BOOL := FALSE;
    Distributed_FailSafe_Consensus_Valid : BOOL := FALSE;

    // Fail-safe conflict detectors.
    CrossDomain_FailSafe_Conflict_Detected : BOOL := FALSE;
    Unsafe_Recovery_Topology_Detected : BOOL := FALSE;
    CrossDomain_Recovery_Race_Detected : BOOL := FALSE;
    Distributed_SafeState_Fork_Detected : BOOL := FALSE;
    PowerDomain_Unsafe_Reactivation_Detected : BOOL := FALSE;
    MultiDomain_Recovery_Deadlock_Detected : BOOL := FALSE;

    // Fail-safe epochs.
    CrossDomain_FailSafe_Closure_Epoch : UDINT := 0;
    CrossDomain_FailSafe_Closure_Epoch_Coherent : BOOL := FALSE;

    // Temporal authority.
    CrossDomain_FailSafe_Closure_Last_Update_MS : UDINT := 0;
    CrossDomain_FailSafe_Closure_Lease_Expired : BOOL := TRUE;

    // Diagnostics.
    CrossDomain_FailSafe_Closure_Last_Error_Code : UDINT := 0;
    CrossDomain_FailSafe_Closure_Last_Error_Text : STRING(160) := '';
    CrossDomain_FailSafe_Closure_Invalidation_Count : UDINT := 0;
END_VAR

(* ---- GVL_DEBUG_VIEW.gvl ---- *)
VAR_GLOBAL
    D_Current_Time_MS : UDINT := 0;

    D_Safety_Mode : E_Safety_Mode := NORMAL;
    D_Safety_Active : BOOL := FALSE;
    D_Recovery_Phase : E_Recovery_Phase := IDLE;
    D_Recovery_Active : BOOL := FALSE;

    D_Current_Scenario : STRING(255) := '';
    D_Behavior_Reason : STRING(255) := '';
    D_Score_Night : INT := 0;
    D_Score_Preheat : INT := 0;
    D_Score_VentBoost : INT := 0;
    D_Score_AccessSecure : INT := 0;
    D_Intent_Night : BOOL := FALSE;
    D_Intent_Comfort : BOOL := FALSE;
    D_Intent_VentBoost : BOOL := FALSE;
    D_Intent_AccessSecure : BOOL := FALSE;

    D_Heating_Block : BOOL := FALSE;
    D_Vent_Stop : BOOL := FALSE;
    D_Water_Block : BOOL := FALSE;
    D_Access_Open_Active : BOOL := FALSE;

    D_Global_Reason : STRING(255) := '';
    D_Behavior_Why_Active : STRING(255) := '';
    D_Heating_Why_Blocked : STRING(255) := '';
    D_Vent_Why_Stopped : STRING(255) := '';
    D_Water_Why_Closed : STRING(255) := '';
    D_Access_Why_Opened : STRING(255) := '';

    D_Main_VentBoost_Zone : INT := 0;
    D_Main_VentBoost_Zone_Weight : REAL := 0.0;
    D_Main_VentBoost_Zone_Confidence : REAL := 0.0;
    D_Max_VentBoost_Zone_Weight : REAL := 0.0;
    D_Min_VentBoost_Zone_Weight : REAL := 0.0;

    // HMI / dashboard sensor quality view.
    D_Input_Source_Valid : BOOL := FALSE;
    D_Input_Degraded : BOOL := FALSE;
    D_Sensor_Fault : BOOL := FALSE;
    D_Validation_Failed : BOOL := FALSE;
    D_Anomaly_Detected : BOOL := FALSE;
    D_Validation_Reason : STRING(120) := '';
    D_Anomaly_Reason : STRING(120) := '';
    D_Last_Invalid_Zone : INT := 0;
    D_Min_Zone_Confidence : REAL := 1.0;
    D_Worst_Zone : INT := 0;

    // Runtime diagnostics formerly stored in legacy GVL_TEST.
    D_Ownership_Violation : BOOL := FALSE;

    D_Adapt_Profile : E_Adapt_Profile := ADAPT_PROFILE_BALANCED;
    D_Adapt_Profile_Text : STRING(32) := 'BALANCED';

    D_Last_Trace_Text : STRING(120) := '';
    D_Last_Trace_Time_MS : UDINT := 0;
    D_Last_Trace_Reason : E_System_Reason_Code := REASON_NONE;
END_VAR

(* ---- GVL_DETERMINISTIC_RECOVERY_PATH_FABRIC.gvl ---- *)
VAR_GLOBAL
    Deterministic_Recovery_Path_Valid : BOOL := FALSE;
    Deterministic_Recovery_Path_Granted : BOOL := FALSE;
    Deterministic_Recovery_Path_Quarantine_Active : BOOL := TRUE;

    Deterministic_Recovery_Path_Canonical : BOOL := FALSE;
    Recovery_Lineage_Causality_Valid : BOOL := FALSE;
    Recovery_Physical_Convergence_Stable : BOOL := FALSE;
    Recovery_Timeline_Monotonic : BOOL := FALSE;

    Recovery_Causality_Grounded : BOOL := FALSE;
    Recovery_Path_Continuity_Valid : BOOL := FALSE;
    Distributed_Recovery_Consensus_Valid : BOOL := FALSE;

    Unsafe_Recovery_Path_Detected : BOOL := FALSE;
    Recovery_Path_Divergence_Detected : BOOL := FALSE;
    Recovery_Causality_Break_Detected : BOOL := FALSE;
    Distributed_Recovery_Fork_Detected : BOOL := FALSE;

    Deterministic_Recovery_Path_Epoch : UDINT := 0;
    Deterministic_Recovery_Path_Last_Update_MS : UDINT := 0;
END_VAR

(* ---- GVL_DISTRIBUTED_EPOCH.gvl ---- *)
VAR_GLOBAL
    // ======================================================
    // DISTRIBUTED EPOCH CONSISTENCY STATE
    // ======================================================
    // Distributed peer epoch reconciliation foundation.
    //
    // Ownership split:
    // - Local_* fields are local authority projections written by
    //   PRG_Distributed_Epoch_Governor.
    // - Peer_* input fields are normalized peer-session projections
    //   written by PRG_Distributed_Peer_Ingestion.
    // - Distributed_* aggregate authority fields are written by
    //   PRG_Distributed_Epoch_Governor.
    //
    // This GVL must not be written by output, verifier, recovery
    // or observability layers.
    // ======================================================

    Distributed_Epoch : ULINT := 0;
    Distributed_Reconciliation_Epoch : ULINT := 0;

    Local_Runtime_Epoch : ULINT := 0;
    Peer_Runtime_Epoch : ULINT := 0;

    Local_Snapshot_Epoch : ULINT := 0;
    Peer_Snapshot_Epoch : ULINT := 0;

    Local_Boot_Generation : ULINT := 0;
    Peer_Boot_Generation : ULINT := 0;

    Local_Fencing_Token : ULINT := 0;
    Peer_Fencing_Token : ULINT := 0;

    Distributed_Epoch_Consistent : BOOL := FALSE;
    Distributed_Reconciliation_Valid : BOOL := FALSE;
    Distributed_Publication_Allowed : BOOL := FALSE;

    Peer_Lease_Active : BOOL := FALSE;
    Peer_Lease_Expired : BOOL := FALSE;
    Peer_Lease_Timeout_MS : UDINT := 5000;

    Peer_Last_Refresh_MS : UDINT := 0;
    Peer_Last_Reconciliation_MS : UDINT := 0;

    Peer_Snapshot_Stale : BOOL := FALSE;
    Peer_Runtime_Stale : BOOL := FALSE;
    Peer_Boot_Mismatch : BOOL := FALSE;
    Peer_Fencing_Conflict : BOOL := FALSE;
    Peer_Semantic_Continuity_Lost : BOOL := FALSE;

    Distributed_Quarantine_Active : BOOL := FALSE;

    Distributed_Last_Error_Code : UDINT := 0;
    Distributed_Last_Error_Text : STRING(160) := '';
END_VAR

(* ---- GVL_DISTRIBUTED_FORWARD_PROGRESS_FABRIC.gvl ---- *)
VAR_GLOBAL
    Distributed_Forward_Progress_Valid : BOOL := FALSE;
    Distributed_Forward_Progress_Granted : BOOL := FALSE;

    Distributed_Forward_Progress_Canonical : BOOL := FALSE;
    Cluster_Progress_Consensus_Stable : BOOL := FALSE;
    Distributed_Recovery_Progress_Valid : BOOL := FALSE;

    Distributed_Progress_Causality_Valid : BOOL := FALSE;
    Cluster_Execution_Lineage_Coherent : BOOL := FALSE;

    Distributed_Livelock_Detected : BOOL := FALSE;
    Cluster_Progress_Fork_Detected : BOOL := FALSE;
    Distributed_Consensus_Progress_Deadlock : BOOL := FALSE;

    Distributed_Forward_Progress_Epoch : UDINT := 0;
END_VAR

(* ---- GVL_Distributed_Projection_Ownership.gvl ---- *)
{attribute 'qualified_only'}
VAR_GLOBAL
    G_Projection_Ownership : ARRAY[1..128] OF ST_Distributed_Projection_Ownership;
END_VAR

VAR_GLOBAL
    G_Runtime_Valid : BOOL;
    G_Last_Update_MS : UDINT;

    G_Any_Ownership_Conflict : BOOL;
    G_Any_Ownership_Stale : BOOL;
    G_Any_Projection_Blocked : BOOL;

    G_Status_Code : UINT;
    G_Status_Text : STRING(160);
END_VAR

(* ---- GVL_DISTRIBUTED_SAFETY_REALITY_CONSENSUS_FABRIC.gvl ---- *)
VAR_GLOBAL
    Distributed_Safety_Reality_Consensus_Valid : BOOL := FALSE;
    Distributed_Safety_Reality_Consensus_Granted : BOOL := FALSE;

    Distributed_Safety_Consensus_Valid : BOOL := FALSE;
    Cluster_Safety_Reality_Stable : BOOL := FALSE;
    Distributed_Observability_Reality_Equivalence : BOOL := FALSE;

    Distributed_Safety_Causality_Valid : BOOL := FALSE;
    Cluster_Safety_Lineage_Coherent : BOOL := FALSE;

    Distributed_Safety_State_Fork : BOOL := FALSE;
    Cluster_Safety_Projection_Drift : BOOL := FALSE;
    Distributed_Unsafe_State_Hidden : BOOL := FALSE;

    Distributed_Safety_Reality_Epoch : UDINT := 0;
END_VAR

(* ---- GVL_ENVIRONMENTAL_AUTHORITY.gvl ---- *)
VAR_GLOBAL
    // Global environmental authority.
    Environmental_Authority_Valid : BOOL := FALSE;
    Environmental_Authority_Granted : BOOL := FALSE;
    Environmental_Quarantine_Active : BOOL := TRUE;

    // Environmental causality proofs.
    External_Environment_Causally_Compatible : BOOL := FALSE;
    Utility_Environment_Stable : BOOL := FALSE;
    Hydraulic_Source_Stable : BOOL := FALSE;
    Thermal_Environment_Stable : BOOL := FALSE;
    Airflow_Environment_Stable : BOOL := FALSE;

    // External environment monitoring.
    Mains_Quality_Valid : BOOL := FALSE;
    Supply_Water_Available : BOOL := FALSE;
    Outdoor_Airflow_Valid : BOOL := FALSE;
    Freeze_Protection_Valid : BOOL := FALSE;

    // Environmental failure prediction.
    Freeze_Front_Propagation_Detected : BOOL := FALSE;
    Utility_Instability_Propagation_Detected : BOOL := FALSE;
    External_Hydraulic_Collapse_Detected : BOOL := FALSE;
    Airflow_Icing_Condition_Detected : BOOL := FALSE;
    Environmental_Rebound_Race_Detected : BOOL := FALSE;

    // Environmental authority epochs.
    Environmental_Authority_Epoch : UDINT := 0;
    Environmental_Authority_Epoch_Coherent : BOOL := FALSE;

    // Temporal environmental authority.
    Environmental_Last_Update_MS : UDINT := 0;
    Environmental_Lease_Expired : BOOL := TRUE;

    // Diagnostics.
    Environmental_Last_Error_Code : UDINT := 0;
    Environmental_Last_Error_Text : STRING(160) := '';
    Environmental_Invalidation_Count : UDINT := 0;
END_VAR

(* ---- GVL_FORENSIC_EVIDENCE_FABRIC.gvl ---- *)
VAR_GLOBAL
    // Global deterministic forensic evidence authority.
    Forensic_Evidence_Valid : BOOL := FALSE;
    Forensic_Evidence_Granted : BOOL := FALSE;
    Forensic_Evidence_Quarantine_Active : BOOL := TRUE;

    // Immutable causality preservation proofs.
    Authority_Lineage_Reconstructable : BOOL := FALSE;
    Decision_Causality_Traceable : BOOL := FALSE;
    Distributed_Evidence_Coherent : BOOL := FALSE;
    Immutable_Audit_Continuity_Valid : BOOL := FALSE;
    Recovery_Lineage_Preserved : BOOL := FALSE;

    // Long-term forensic integrity.
    Historical_Proof_Chain_Valid : BOOL := FALSE;
    Governance_Event_Lineage_Coherent : BOOL := FALSE;
    Semantic_Transition_Traceable : BOOL := FALSE;
    Physical_Transition_Traceable : BOOL := FALSE;

    // Forensic split-brain detectors.
    Authority_Lineage_Gap_Detected : BOOL := FALSE;
    NonReconstructable_Decision_Detected : BOOL := FALSE;
    History_Evidence_Divergence_Detected : BOOL := FALSE;
    Causal_Chain_Erosion_Detected : BOOL := FALSE;
    Distributed_Forensic_Inconsistency_Detected : BOOL := FALSE;
    Immutable_Audit_Discontinuity_Detected : BOOL := FALSE;

    // Forensic epochs.
    Forensic_Evidence_Epoch : UDINT := 0;
    Forensic_Evidence_Epoch_Coherent : BOOL := FALSE;

    // Temporal authority.
    Forensic_Evidence_Last_Update_MS : UDINT := 0;
    Forensic_Evidence_Lease_Expired : BOOL := TRUE;

    // Diagnostics.
    Forensic_Evidence_Last_Error_Code : UDINT := 0;
    Forensic_Evidence_Last_Error_Text : STRING(160) := '';
    Forensic_Evidence_Invalidation_Count : UDINT := 0;
END_VAR

(* ---- GVL_GATEWAY.gvl ---- *)
{attribute 'qualified_only'}
VAR_GLOBAL
    G_Gateway_Command : ST_Gateway_Command;
    G_Gateway_Command_Received : BOOL;
    G_Gateway_Send_2FA : BOOL;
    G_Gateway_2FA_Code : STRING(6);
    G_Gateway_Telegram_Msg : STRING(200);
    G_Gateway_Send_Telegram : BOOL;
    G_Gateway_HMI_Status_Message : STRING(200);
    G_Gateway_Ping_OK : BOOL;
    G_Gateway_Data_Ready : BOOL;
    G_Gateway_Modbus_Registers : ARRAY[0..GVL_CONSTANTS.C_MAX_MODBUS_REGISTERS-1] OF WORD;

    // === SHADOW POLICY EXPORT ===
    G_Shadow_Alert_Active : BOOL;
    G_Shadow_Dominant_Channel : STRING(32);
    G_Shadow_Policy_Summary_Text : STRING(160);
    G_Shadow_Recent_Activity_Text : STRING(160);
    G_Shadow_Rate_Summary_Text : STRING(160);
    G_Shadow_Total_Fallback_Count : UDINT;
    G_Shadow_Total_Recovery_Count : UDINT;
END_VAR

(* ---- GVL_GOVERNANCE_LIVENESS_INTEGRITY_FABRIC.gvl ---- *)
VAR_GLOBAL
    // Deterministic governance liveness integrity governance.
    Governance_Liveness_Integrity_Valid : BOOL := FALSE;
    Governance_Liveness_Integrity_Granted : BOOL := FALSE;
    Governance_Liveness_Integrity_Quarantine_Active : BOOL := TRUE;

    // Governance execution liveness proofs.
    Governance_Execution_Liveness_Stable : BOOL := FALSE;
    Integrity_Governor_Scheduling_Canonical : BOOL := FALSE;
    CrossGovernor_Execution_Continuity_Valid : BOOL := FALSE;
    Deterministic_Validation_Cycle_Integrity : BOOL := FALSE;
    Governance_Runtime_Liveness_Coherent : BOOL := FALSE;

    // Runtime scheduling integrity.
    Validation_Cycle_Timing_Monotonic : BOOL := FALSE;
    Distributed_Governor_Execution_Aligned : BOOL := FALSE;
    Runtime_Integrity_Causality_Grounded : BOOL := FALSE;
    Governance_Execution_Budget_Stable : BOOL := FALSE;

    // Governance liveness degradation detectors.
    Integrity_Governor_Starvation_Detected : BOOL := FALSE;
    Validation_Cycle_Skip_Detected : BOOL := FALSE;
    CrossGovernor_Execution_Jitter_Fork : BOOL := FALSE;
    Selective_Governance_Degradation_Detected : BOOL := FALSE;
    Runtime_Governor_Execution_Stall_Detected : BOOL := FALSE;
    Distributed_Liveness_Reality_Fork_Detected : BOOL := FALSE;

    // Liveness epochs.
    Governance_Liveness_Integrity_Epoch : UDINT := 0;
    Governance_Liveness_Integrity_Epoch_Coherent : BOOL := FALSE;

    // Temporal authority.
    Governance_Liveness_Integrity_Last_Update_MS : UDINT := 0;
    Governance_Liveness_Integrity_Lease_Expired : BOOL := TRUE;

    // Diagnostics.
    Governance_Liveness_Integrity_Last_Error_Code : UDINT := 0;
    Governance_Liveness_Integrity_Last_Error_Text : STRING(160) := '';
    Governance_Liveness_Integrity_Invalidation_Count : UDINT := 0;
END_VAR

(* ---- GVL_GOVERNANCE_OBSERVER_CONSENSUS_FABRIC.gvl ---- *)
VAR_GLOBAL
    // Deterministic governance observer consensus governance.
    Governance_Observer_Consensus_Valid : BOOL := FALSE;
    Governance_Observer_Consensus_Granted : BOOL := FALSE;
    Governance_Observer_Consensus_Quarantine_Active : BOOL := TRUE;

    // Distributed governance projection proofs.
    Distributed_Governance_Projection_Consistent : BOOL := FALSE;
    Observer_Semantic_Consensus_Valid : BOOL := FALSE;
    CrossNode_Authority_Interpretation_Aligned : BOOL := FALSE;
    Governance_Reality_Canonical : BOOL := FALSE;
    Observer_Projection_Lineage_Coherent : BOOL := FALSE;

    // Observer consensus integrity.
    Canonical_Projection_Vector_Stable : BOOL := FALSE;
    Distributed_Interpretation_Equivalence_Valid : BOOL := FALSE;
    Governance_Projection_Causality_Grounded : BOOL := FALSE;
    Observer_Timeline_Consensus_Monotonic : BOOL := FALSE;

    // Governance observer split-brain detectors.
    Observer_Governance_Divergence_Detected : BOOL := FALSE;
    CrossNode_Authority_Interpretation_Fork : BOOL := FALSE;
    Semantic_Projection_Mismatch_Detected : BOOL := FALSE;
    Canonical_Governance_Reality_Lost : BOOL := FALSE;
    Observer_Projection_Lineage_Drift_Detected : BOOL := FALSE;
    Distributed_Governance_Reality_Fork_Detected : BOOL := FALSE;

    // Consensus epochs.
    Governance_Observer_Consensus_Epoch : UDINT := 0;
    Governance_Observer_Consensus_Epoch_Coherent : BOOL := FALSE;

    // Temporal authority.
    Governance_Observer_Consensus_Last_Update_MS : UDINT := 0;
    Governance_Observer_Consensus_Lease_Expired : BOOL := TRUE;

    // Diagnostics.
    Governance_Observer_Consensus_Last_Error_Code : UDINT := 0;
    Governance_Observer_Consensus_Last_Error_Text : STRING(160) := '';
    Governance_Observer_Consensus_Invalidation_Count : UDINT := 0;
END_VAR

(* ---- GVL_HEALTH_BRIDGE.gvl ---- *)
{attribute 'qualified_only'}
VAR_GLOBAL
    G_Smoke_Detected : BOOL;
    G_Gas_Detected : BOOL;
    G_Leak_Detected : BOOL;
    G_Leak_Warning_Level : BOOL;
    G_CO_Warning_Level : BOOL;
    G_CO_Alarm_Level : BOOL;
    G_Last_Fault_Event_Text : STRING(255);
    G_Role_Conflict_Error : BOOL;
END_VAR

(* ---- GVL_Heating_Runtime_Explainability.gvl ---- *)
{attribute 'qualified_only'}
VAR_GLOBAL
    // Passive runtime explainability publication surface.
    // Observation-only: no command, output or runtime authority.
    G_Runtime_Phase_Event : ST_Heating_Runtime_Phase_Event;
    G_Runtime_Anomaly : ST_Heating_Runtime_Anomaly;
    G_Runtime_Blackbox_Event : ST_Heating_Runtime_Blackbox_Event;
    G_Runtime_Blackbox_Timeline : ST_Heating_Runtime_Blackbox_Timeline;
    G_Runtime_Event_Buffer : ST_Heating_Runtime_Event_Buffer;
    G_Runtime_Adaptive_Intelligence : ST_Heating_Runtime_Adaptive_Intelligence;
    G_Runtime_Causality_Graph : ST_Heating_Runtime_Causality_Graph;
    G_Runtime_Integration_Bridge : ST_Heating_Runtime_Integration_Bridge;
    G_Runtime_Predictive_State : ST_Heating_Runtime_Predictive_State;
    G_Runtime_Execution_Timeline : ST_Heating_Runtime_Execution_Timeline;
    G_Runtime_Phase_Transition : ST_Heating_Runtime_Phase_Transition;

    G_Runtime_Explainability_Publication_Valid : BOOL := FALSE;
    G_Runtime_Explainability_Status_Code : UINT := 0;
    G_Runtime_Explainability_Status_Text : STRING(128) := 'Heating runtime explainability inactive';
END_VAR

(* ---- GVL_Heating_Runtime_Supervisory_Publication.gvl ---- *)
{attribute 'qualified_only'}
VAR_GLOBAL
    // Canonical supervisory publication surface.
    // Runtime-independent passive observability publication.

    G_Publication : ST_Heating_Runtime_Supervisory_Publication;
END_VAR

(* ---- GVL_HISTORICAL_ORDERING_INTEGRITY_FABRIC.gvl ---- *)
VAR_GLOBAL
    Historical_Ordering_Integrity_Valid : BOOL := FALSE;
    Historical_Ordering_Integrity_Granted : BOOL := FALSE;

    Historical_Ordering_Integrity_Granted_Proof : BOOL := FALSE;
    Historical_Timeline_Canonical : BOOL := FALSE;
    Forensic_Ordering_Coherent : BOOL := FALSE;

    Historical_Causality_Grounded : BOOL := FALSE;
    Distributed_Historical_Consensus_Valid : BOOL := FALSE;

    Historical_Order_Divergence : BOOL := FALSE;
    Unsafe_Historical_Rewrite_Detected : BOOL := FALSE;
    Historical_Causality_Gap_Detected : BOOL := FALSE;

    Historical_Ordering_Epoch : UDINT := 0;
END_VAR

(* ---- GVL_HMI.gvl ---- *)
{attribute 'qualified_only'}
VAR_GLOBAL
    // Heating dashboard
    G_HMI_Heating_Confidence : REAL := 1.0;
    G_HMI_Heating_Confidence_Percent : INT := 100;
    G_HMI_Heating_Reason_Code : INT := 0;
    G_HMI_Heating_Status_Text : STRING(128) := 'OK';
    G_HMI_Heating_Status_Level : INT := 0; // 0=OK, 1=WARN, 2=ALARM

    // Heating cascade dashboard
    G_HMI_Heating_Cascade_Available : BOOL;
    G_HMI_Heating_Cascade_Degraded : BOOL;
    G_HMI_Heating_Cascade_Partial_Capacity : BOOL;
    G_HMI_Heating_Cascade_No_Flame : BOOL;
    G_HMI_Heating_Cascade_Transport_Degraded : BOOL;
    G_HMI_Heating_Cascade_Ignition_Timeout : BOOL;
    G_HMI_Heating_Cascade_Active_Boilers : UINT;
    G_HMI_Heating_Cascade_Available_Boilers : UINT;

    // OpenTherm dashboard
    G_HMI_Boiler_OT_Online : ARRAY[1..GVL_CONSTANTS.C_MAX_BOILERS] OF BOOL;
    G_HMI_Boiler_OT_Command_Ack : ARRAY[1..GVL_CONSTANTS.C_MAX_BOILERS] OF BOOL;
    G_HMI_Boiler_OT_Command_Timeout : ARRAY[1..GVL_CONSTANTS.C_MAX_BOILERS] OF BOOL;
    G_HMI_Boiler_OT_Heartbeat_Timeout : ARRAY[1..GVL_CONSTANTS.C_MAX_BOILERS] OF BOOL;
    G_HMI_Boiler_OT_Adapter_Error : ARRAY[1..GVL_CONSTANTS.C_MAX_BOILERS] OF BOOL;
    G_HMI_Boiler_OT_Heartbeat_Age_MS : ARRAY[1..GVL_CONSTANTS.C_MAX_BOILERS] OF UDINT;
    G_HMI_Boiler_OT_Command_Age_MS : ARRAY[1..GVL_CONSTANTS.C_MAX_BOILERS] OF UDINT;
    G_HMI_Boiler_OT_Adapter_State : ARRAY[1..GVL_CONSTANTS.C_MAX_BOILERS] OF E_OpenTherm_Adapter_State;
    G_HMI_Boiler_OT_Error_State : ARRAY[1..GVL_CONSTANTS.C_MAX_BOILERS] OF E_OpenTherm_Error;

    // Heating predictive dashboard
    G_HMI_Heating_Predictive_Pressure_Drop : ARRAY[1..GVL_CONSTANTS.C_MAX_MANIFOLDS] OF BOOL;
    G_HMI_Heating_Predictive_Current_Rise : ARRAY[1..GVL_CONSTANTS.C_MAX_MANIFOLDS] OF BOOL;
END_VAR

(* ---- GVL_INDUSTRIAL_MAINTAINABILITY_FABRIC.gvl ---- *)
VAR_GLOBAL
    // Industrial maintainability governance.
    Industrial_Maintainability_Active : BOOL := TRUE;
    Industrial_Maintainability_ReadOnly : BOOL := TRUE;

    // Runtime heat mapping.
    Verification_Runtime_Heat_Observed : BOOL := FALSE;
    Diagnostics_Runtime_Heat_Observed : BOOL := FALSE;
    Observability_Runtime_Heat_Observed : BOOL := FALSE;
    Governance_Runtime_Heat_Observed : BOOL := FALSE;

    // Semantic dead-code and fossilization observations.
    Unused_Semantic_Pathways_Observed : BOOL := FALSE;
    Inactive_Governance_Chains_Observed : BOOL := FALSE;
    NonContributing_Verification_Layers_Observed : BOOL := FALSE;
    Semantic_Fossilization_Risk : BOOL := FALSE;

    // Semantic freeze boundary.
    Semantic_Freeze_Boundary_Active : BOOL := TRUE;
    New_Semantic_Layers_Restricted : BOOL := FALSE;
    Survivability_Justification_Required : BOOL := TRUE;

    // Maintainability pressure.
    Merge_Conflict_Risk_Observed : BOOL := FALSE;
    Audit_Complexity_Pressure_Observed : BOOL := FALSE;
    Maintenance_Entropy_Observed : BOOL := FALSE;

    Industrial_Maintainability_Epoch : UDINT := 0;
END_VAR

(* ---- GVL_INPUT.gvl ---- *)
VAR_GLOBAL
    IN_Last_Update_MS : UDINT := 0;
    IN_Source_Valid : BOOL := FALSE;

    IN_Room_Temps : ARRAY[1..GVL_CONSTANTS.C_MAX_ZONES] OF REAL;
    IN_Floor_Temps : ARRAY[1..GVL_CONSTANTS.C_MAX_HEATING_CIRCUITS] OF REAL;
    IN_Room_Hum : ARRAY[1..GVL_CONSTANTS.C_MAX_ZONES] OF REAL;
    IN_Room_CO2 : ARRAY[1..GVL_CONSTANTS.C_MAX_ZONES] OF REAL;

    IN_Outdoor_Temp : REAL := 0.0;
    IN_Preheat_Request : BOOL := FALSE;
    IN_Freeze_Request : BOOL := FALSE;

    IN_Water_Sensors : ARRAY[1..GVL_CONSTANTS.C_MAX_FLOOD_SENSORS] OF BOOL;
    IN_Smoke_Sensors : ARRAY[1..GVL_CONSTANTS.C_MAX_SMOKE_SENSORS] OF BOOL;
    IN_Methane_Sensors : ARRAY[1..GVL_CONSTANTS.C_MAX_METHANE_SENSORS] OF REAL;
    IN_CO_Sensors : ARRAY[1..GVL_CONSTANTS.C_MAX_CO_SENSORS] OF REAL;

    IN_Input_Degraded : BOOL := FALSE;
    IN_Sensor_Fault : BOOL := FALSE;

    IN_Validation_Failed : BOOL := FALSE;
    IN_Anomaly_Detected : BOOL := FALSE;
    IN_Validation_Reason : STRING(120) := '';
    IN_Anomaly_Reason : STRING(120) := '';
    IN_Last_Invalid_Zone : INT := 0;

    IN_Room_Temp_Prev : ARRAY[1..GVL_CONSTANTS.C_MAX_ZONES] OF REAL;
    IN_Room_Hum_Prev : ARRAY[1..GVL_CONSTANTS.C_MAX_ZONES] OF REAL;
    IN_Last_Change_MS : ARRAY[1..GVL_CONSTANTS.C_MAX_ZONES] OF UDINT;

    IN_Room_Temp_Confidence : ARRAY[1..GVL_CONSTANTS.C_MAX_ZONES] OF REAL;
    IN_Room_Hum_Confidence : ARRAY[1..GVL_CONSTANTS.C_MAX_ZONES] OF REAL;
    IN_Zone_Confidence : ARRAY[1..GVL_CONSTANTS.C_MAX_ZONES] OF REAL;

    // NEW: reputation (long-term learning)
    IN_Room_Temp_Reputation : ARRAY[1..GVL_CONSTANTS.C_MAX_ZONES] OF REAL;
    IN_Room_Hum_Reputation : ARRAY[1..GVL_CONSTANTS.C_MAX_ZONES] OF REAL;

    IN_Min_Zone_Confidence : REAL := 1.0;
    IN_Worst_Zone : INT := 0;
END_VAR

(* ---- GVL_INPUT_QUALITY.gvl ---- *)
VAR_GLOBAL
    G_Room_Temp_Quality : ARRAY[1..16] OF ST_Input_Quality_Record;
    G_Floor_Temp_Quality : ARRAY[1..GVL_CONSTANTS.C_MAX_HEATING_CIRCUITS] OF ST_Input_Quality_Record;
END_VAR

(* ---- GVL_IO.gvl ---- *)
{attribute 'qualified_only'}
VAR_GLOBAL
    // ======================================================
    // PHYSICAL IO SURFACE
    // ======================================================
    // Input fields are hardware/mapping observations.
    // Output fields are the terminal physical publication surface.
    //
    // PRG_IO_Write is the only runtime-layer publisher for physical
    // output commands in this GVL. Upstream authority/governance,
    // verifier, recovery and observability layers must not write
    // physical outputs directly.
    // ======================================================

    DI_Security_Open : ARRAY[1..GVL_CONSTANTS.C_MAX_SECURITY_SENSORS] OF BOOL;
    DI_Security_Glass : ARRAY[1..GVL_CONSTANTS.C_MAX_SECURITY_SENSORS] OF BOOL;
    DI_Security_2F_Group : BOOL;
    DI_Flood_Sensors : ARRAY[1..GVL_CONSTANTS.C_MAX_FLOOD_SENSORS] OF BOOL;
    DI_Manifold_End_Switches : ARRAY[1..GVL_CONSTANTS.C_MAX_MANIFOLDS] OF BOOL;
    AO_Manifold_Valves : ARRAY[1..GVL_CONSTANTS.C_MAX_MANIFOLDS] OF UINT;
    DO_Manifold_Pumps : ARRAY[1..GVL_CONSTANTS.C_MAX_MANIFOLDS] OF BOOL;
    AI_Manifold_Currents : ARRAY[1..GVL_CONSTANTS.C_MAX_MANIFOLDS] OF INT;
    AI_Manifold_Pressures : ARRAY[1..GVL_CONSTANTS.C_MAX_MANIFOLDS] OF INT;
    AI_Manifold_Temps_Supply : ARRAY[1..GVL_CONSTANTS.C_MAX_MANIFOLDS] OF ST_Owen_Analog_Value;
    AI_Manifold_Temps_Return : ARRAY[1..GVL_CONSTANTS.C_MAX_MANIFOLDS] OF INT;
    AO_Supply_Fans : ARRAY[1..GVL_CONSTANTS.C_MAX_SUPPLY_FANS] OF UINT;
    AO_Exhaust_Fans : ARRAY[1..GVL_CONSTANTS.C_MAX_EXHAUST_FANS] OF UINT;
    AO_Lighting_Levels : ARRAY[1..GVL_CONSTANTS.C_MAX_LIGHT_ZONES] OF UINT;
    AO_Blinds_Positions : ARRAY[1..GVL_CONSTANTS.C_MAX_BLINDS] OF UINT;
    AI_Supply_Temps : ARRAY[1..GVL_CONSTANTS.C_MAX_SUPPLY_TEMPS] OF ST_Owen_Analog_Value;
    AI_Boiler_Modulation : ARRAY[1..GVL_CONSTANTS.C_MAX_BOILERS] OF INT;
    AI_Boiler_Flame_Status : ARRAY[1..GVL_CONSTANTS.C_MAX_BOILERS] OF BOOL;
    DI_Boiler_Error : ARRAY[1..GVL_CONSTANTS.C_MAX_BOILERS] OF BOOL;
    AI_Methane_LEL : ARRAY[1..GVL_CONSTANTS.C_MAX_METHANE_SENSORS] OF ST_Owen_Analog_Value;
    AI_CO_PPM : ARRAY[1..GVL_CONSTANTS.C_MAX_CO_SENSORS] OF REAL;
    DI_Smoke_Sensors : ARRAY[1..GVL_CONSTANTS.C_MAX_SMOKE_SENSORS] OF BOOL;
    AI_Temp_Outdoor : ST_Owen_Analog_Value;
    AI_Floor_Temps : ARRAY[1..GVL_CONSTANTS.C_MAX_ZONES] OF REAL;
    AI_Room_Temps : ARRAY[1..GVL_CONSTANTS.C_MAX_ZONES] OF REAL;
    AI_Room_Hum : ARRAY[1..GVL_CONSTANTS.C_MAX_ZONES] OF REAL;
    AI_Room_CO2 : ARRAY[1..GVL_CONSTANTS.C_MAX_ZONES] OF REAL;
    DO_Zone_Valves : ARRAY[1..GVL_CONSTANTS.C_MAX_HEATING_CIRCUITS] OF BOOL;
    AI_DHW_Temp : REAL;
    AI_DHW_Pressure : REAL;
    DO_DHW_Heating_Pump : BOOL;
    DO_DHW_Circ_Pump : BOOL;
    DO_Backup_Circulation_Pump : BOOL;
    DO_Electric_Heater_Enable : BOOL;
    DI_Lighting_Switches : ARRAY[1..GVL_CONSTANTS.C_MAX_LIGHT_ZONES] OF BOOL;
    DI_Socket_Switches : ARRAY[1..GVL_CONSTANTS.C_MAX_SOCKETS] OF BOOL;
    DI_Motion_Sensors : ARRAY[1..GVL_CONSTANTS.C_MAX_LIGHT_ZONES] OF BOOL;
    DO_Sockets : ARRAY[1..GVL_CONSTANTS.C_MAX_SOCKETS] OF BOOL;
    DO_Gas_Valve_Close : BOOL;
    DO_Water_Valve_35_Close : BOOL;
    DO_Water_Valve_36_Close : BOOL;
    AI_Water_Valve_35_Current : REAL;
    AI_Water_Valve_36_Current : REAL;
    DI_Power_OK : BOOL;
    DO_Gas_Siren : BOOL;
    DO_Fire_Siren : BOOL;
    DO_Security_Siren : BOOL;
    DO_Pump_Main_Enable : BOOL;
    DO_Gate_Open : BOOL;
    DO_Wicket_Open : BOOL;
    DO_Lock_1_Open : BOOL;
    DO_Lock_1_Close : BOOL;
    DO_Lock_2_Open : BOOL;
    DO_Lock_2_Close : BOOL;
    DI_Partner_Pulse : BOOL;
    DI_Partner_Active : BOOL;
    DO_Heartbeat_Pulse : BOOL;
    DO_Active_Status : BOOL;
    DI_Module_1_Heartbeat : BOOL;
    DI_Module_2_Heartbeat : BOOL;
    DI_Backup_Circulation_Pump_Feedback : BOOL;
    DI_Electric_Heater_Feedback : BOOL;
    DI_Water_Zone_Open_FB : ARRAY[1..GVL_CONSTANTS.C_MAX_WATER_ZONES] OF BOOL;
    DI_Water_Zone_Close_FB : ARRAY[1..GVL_CONSTANTS.C_MAX_WATER_ZONES] OF BOOL;
    DO_Water_Zone_Enable : ARRAY[1..GVL_CONSTANTS.C_MAX_WATER_ZONES] OF BOOL;
END_VAR

(* ---- GVL_IO_Binding_Runtime.gvl ---- *)
{attribute 'qualified_only'}
VAR_GLOBAL
    G_Flood_Sensor_Value : ARRAY[1..64] OF BOOL;
    G_Flood_Sensor_Valid : ARRAY[1..64] OF BOOL;

    G_Water_Valve_Open_FB_Value : ARRAY[1..64] OF BOOL;
    G_Water_Valve_Open_FB_Valid : ARRAY[1..64] OF BOOL;

    G_Water_Valve_Close_FB_Value : ARRAY[1..64] OF BOOL;
    G_Water_Valve_Close_FB_Valid : ARRAY[1..64] OF BOOL;

    G_Water_Valve_Output_Channel_Valid : ARRAY[1..64] OF BOOL;

    G_Runtime_Valid : BOOL;
    G_Last_Update_MS : UDINT;

    G_Any_Invalid_Binding : BOOL;
    G_Any_Missing_Binding : BOOL;

    G_Status_Code : UINT;
    G_Status_Text : STRING(128);
END_VAR

(* ---- GVL_META_GOVERNANCE_FABRIC.gvl ---- *)
VAR_GLOBAL
    // Global deterministic meta-governance authority.
    Meta_Governance_Valid : BOOL := FALSE;
    Meta_Governance_Granted : BOOL := FALSE;
    Meta_Governance_Quarantine_Active : BOOL := TRUE;

    // Recursive governance consistency proofs.
    Governance_Graph_Acyclic : BOOL := FALSE;
    Authority_Rooting_Valid : BOOL := FALSE;
    Independent_Validation_Preserved : BOOL := FALSE;
    Meta_Consistency_Coherent : BOOL := FALSE;
    Recursive_Trust_Boundaries_Stable : BOOL := FALSE;

    // Governance graph integrity.
    Validator_Independence_Valid : BOOL := FALSE;
    CrossLayer_Causality_Grounded : BOOL := FALSE;
    Bootstrap_Validation_Absent : BOOL := FALSE;
    SelfReference_Elimination_Valid : BOOL := FALSE;

    // Meta-governance recursion detectors.
    Recursive_Authority_Dependency_Detected : BOOL := FALSE;
    Circular_Validation_Chain_Detected : BOOL := FALSE;
    SelfJustifying_Governance_State_Detected : BOOL := FALSE;
    Epistemic_Recursion_Leakage_Detected : BOOL := FALSE;
    Authority_Bootstrap_Paradox_Detected : BOOL := FALSE;
    Meta_Consistency_Erosion_Detected : BOOL := FALSE;

    // Governance epochs.
    Meta_Governance_Epoch : UDINT := 0;
    Meta_Governance_Epoch_Coherent : BOOL := FALSE;

    // Temporal authority.
    Meta_Governance_Last_Update_MS : UDINT := 0;
    Meta_Governance_Lease_Expired : BOOL := TRUE;

    // Diagnostics.
    Meta_Governance_Last_Error_Code : UDINT := 0;
    Meta_Governance_Last_Error_Text : STRING(160) := '';
    Meta_Governance_Invalidation_Count : UDINT := 0;
END_VAR

(* ---- GVL_MODBUS_RTU_FRAME.gvl ---- *)
{attribute 'qualified_only'}
VAR_GLOBAL
    // ======================================================
    // MODBUS RTU FRAME RUNTIME
    // ======================================================
    // TX_Frame is built from a confirmed bridge request.
    // RX_Frame is filled only by a concrete serial/RTU driver after physical receive.

    G_TX_Frame : ST_Modbus_RTU_Frame;
    G_RX_Frame : ST_Modbus_RTU_Frame;

    G_TX_Ready : BOOL := FALSE;
    G_RX_Ready : BOOL := FALSE;
    G_Last_TX_MS : UDINT := 0;
    G_Last_RX_MS : UDINT := 0;
END_VAR

(* ---- GVL_OPERATIONAL_INTELLIGENCE_FABRIC.gvl ---- *)
VAR_GLOBAL
    Operational_Intelligence_Active : BOOL := TRUE;
    Operational_Intelligence_ReadOnly : BOOL := TRUE;
    Operational_Intelligence_NoMutation : BOOL := TRUE;

    Dominant_Instability_Source_Available : BOOL := FALSE;
    Active_Degradation_Cause_Available : BOOL := FALSE;
    Recovery_Blocker_Observed : BOOL := FALSE;
    Governance_Pressure_Hotspot_Observed : BOOL := FALSE;

    Operational_Reasoning_Consistency_Valid : BOOL := FALSE;
    Runtime_Causal_Projection_Valid : BOOL := FALSE;
    Distributed_Operational_Context_Valid : BOOL := FALSE;

    Governance_Saturation_Observed : BOOL := FALSE;
    Governance_Complexity_Pressure_Observed : BOOL := FALSE;
    Operational_Opacity_Observed : BOOL := FALSE;

    Operational_Intelligence_Epoch : UDINT := 0;
END_VAR

(* ---- GVL_PERSISTENT.gvl ---- *)
VAR_GLOBAL PERSISTENT RETAIN

    // === SYSTEM ===
    P_System_Mode : E_System_Operating_Mode;

    // === SAFETY LATCHES ===
    P_Safety_Gas_Latched : BOOL;
    P_Safety_Smoke_Latched : BOOL;
    P_Safety_Leak_Latched : BOOL;

    // === HEATING / DHW ===
    P_DHW_Heating_Active : BOOL;

    // === CONTROL ===
    P_Valid : BOOL;

END_VAR

(* ---- GVL_PHYSICAL_SAFETY_PROJECTION_FABRIC.gvl ---- *)
VAR_GLOBAL
    Physical_Safety_Projection_Valid : BOOL := FALSE;
    Physical_Safety_Projection_Granted : BOOL := FALSE;

    Physical_Plant_Safety_Projection_Stable : BOOL := FALSE;
    Energy_State_Safety_Projection_Valid : BOOL := FALSE;
    Recovery_State_Safety_Projection_Valid : BOOL := FALSE;

    Physical_Projection_Causality_Valid : BOOL := FALSE;
    Projection_Reality_Alignment_Stable : BOOL := FALSE;

    Physical_Safety_Projection_Drift_Detected : BOOL := FALSE;
    Hidden_Unsafe_Physical_State_Detected : BOOL := FALSE;
    Unsafe_Projection_Backfill_Detected : BOOL := FALSE;

    Physical_Safety_Projection_Epoch : UDINT := 0;
END_VAR

(* ---- GVL_PHYSICAL_SNAPSHOT.gvl ---- *)
VAR_GLOBAL
    // Immutable physical snapshot authority.
    Physical_Snapshot_Valid : BOOL := FALSE;
    Physical_Snapshot_Frozen : BOOL := FALSE;
    Physical_Snapshot_Publication_Allowed : BOOL := FALSE;
    Physical_Snapshot_Isolation_Valid : BOOL := FALSE;
    Physical_Snapshot_Copy_Valid : BOOL := FALSE;

    // Snapshot epoch coherence.
    Physical_Snapshot_Epoch : UDINT := 0;
    Physical_Snapshot_Runtime_Epoch : UDINT := 0;
    Physical_Snapshot_Output_Epoch : UDINT := 0;

    // Mutation protection.
    Physical_Snapshot_Mutation_Detected : BOOL := FALSE;
    Physical_Snapshot_Replay_Suspected : BOOL := FALSE;
    Physical_Snapshot_Lease_Expired : BOOL := TRUE;

    // Cross-governor coherence.
    Physical_Snapshot_Consensus_Coherent : BOOL := FALSE;
    Physical_Snapshot_Causality_Coherent : BOOL := FALSE;

    // Temporal authority.
    Physical_Snapshot_Last_Update_MS : UDINT := 0;
    Physical_Snapshot_Freshness_Valid : BOOL := FALSE;

    // Diagnostics.
    Physical_Snapshot_Last_Error_Code : UDINT := 0;
    Physical_Snapshot_Last_Error_Text : STRING(160) := '';
    Physical_Snapshot_Invalidation_Count : UDINT := 0;
END_VAR

(* ---- GVL_PHYSICAL_TRANSACTION.gvl ---- *)
VAR_GLOBAL
    // Global physical transaction authority.
    Physical_Transaction_Valid : BOOL := FALSE;
    Physical_Transaction_Granted : BOOL := FALSE;
    Physical_Transaction_Quarantine_Active : BOOL := TRUE;

    // Transaction epochs.
    Physical_Transaction_Epoch : UDINT := 0;
    Physical_Transaction_Command_Epoch : UDINT := 0;
    Physical_Transaction_ACK_Epoch : UDINT := 0;

    // Cross-actuator convergence.
    All_Actuators_Converged : BOOL := FALSE;
    Cross_Actuator_Epoch_Coherent : BOOL := FALSE;
    Distributed_Actuation_Coherent : BOOL := FALSE;
    Stable_Plant_State_Confirmed : BOOL := FALSE;

    // Transaction sequencing.
    Valve_Transition_Confirmed : BOOL := FALSE;
    Pump_Transition_Confirmed : BOOL := FALSE;
    Damper_Transition_Confirmed : BOOL := FALSE;
    Relay_Bank_Transition_Confirmed : BOOL := FALSE;

    // Physical convergence proofs.
    Flow_Stabilization_Confirmed : BOOL := FALSE;
    Pressure_Stabilization_Confirmed : BOOL := FALSE;
    Thermal_Response_Confirmed : BOOL := FALSE;
    Electrical_Load_Stabilized : BOOL := FALSE;

    // Failure/skew detection.
    Partial_Plant_Transition_Detected : BOOL := FALSE;
    Cross_Actuator_Convergence_Skew : BOOL := FALSE;
    Pump_Valve_Ordering_Race_Detected : BOOL := FALSE;
    Distributed_Actuator_Rollback_Detected : BOOL := FALSE;
    Transaction_Timeout_Detected : BOOL := FALSE;
    Brownout_Partial_Switching_Detected : BOOL := FALSE;

    // Temporal authority.
    Physical_Transaction_Last_Update_MS : UDINT := 0;
    Physical_Transaction_Lease_Expired : BOOL := TRUE;

    // Diagnostics.
    Physical_Transaction_Last_Error_Code : UDINT := 0;
    Physical_Transaction_Last_Error_Text : STRING(160) := '';
    Physical_Transaction_Invalidation_Count : UDINT := 0;
END_VAR

(* ---- GVL_PROOF_CONTINUITY_AUDIT_FABRIC.gvl ---- *)
VAR_GLOBAL
    Proof_Continuity_Audit_Active : BOOL := TRUE;

    Proof_Continuity_Observed : BOOL := FALSE;
    Proof_Lineage_Coherent : BOOL := FALSE;
    Proof_Historical_Integrity_Observed : BOOL := FALSE;

    Proof_Audit_ReadOnly_Mode : BOOL := TRUE;
    Proof_Audit_NoTopologyMutation : BOOL := TRUE;

    Proof_Gap_Observed : BOOL := FALSE;
    Proof_Lineage_Drift_Observed : BOOL := FALSE;
    Proof_Consistency_Decay_Observed : BOOL := FALSE;

    Proof_Continuity_Audit_Epoch : UDINT := 0;
END_VAR

(* ---- GVL_PROVENANCE_CONTINUITY_FABRIC.gvl ---- *)
VAR_GLOBAL
    // Deterministic provenance continuity governance.
    Provenance_Continuity_Valid : BOOL := FALSE;
    Provenance_Continuity_Granted : BOOL := FALSE;
    Provenance_Continuity_Quarantine_Active : BOOL := TRUE;

    // Recovery provenance continuity proofs.
    Recovery_Provenance_Reattested : BOOL := FALSE;
    Authority_Resurrection_Authentic : BOOL := FALSE;
    Federation_Rejoin_Provenance_Valid : BOOL := FALSE;
    PostRecovery_TrustSeed_Coherent : BOOL := FALSE;
    CrossEpoch_Provenance_Continuity_Stable : BOOL := FALSE;

    // Recovery trust continuity integrity.
    Recovery_Epoch_Authenticity_Valid : BOOL := FALSE;
    Distributed_Rejoin_Attestation_Coherent : BOOL := FALSE;
    Authority_Restoration_Provenance_Grounded : BOOL := FALSE;
    Provenance_Lease_Continuity_Valid : BOOL := FALSE;

    // Post-recovery provenance bypass detectors.
    Stale_Provenance_Resurrection_Detected : BOOL := FALSE;
    Recovered_Authority_Without_Reattestation_Detected : BOOL := FALSE;
    Federation_Rejoin_Without_Provenance_Detected : BOOL := FALSE;
    CrossEpoch_Trust_Continuity_Broken : BOOL := FALSE;
    Recovery_Trust_Seed_Drift_Detected : BOOL := FALSE;
    Provenance_Resurrection_Bypass_Detected : BOOL := FALSE;

    // Continuity epochs.
    Provenance_Continuity_Epoch : UDINT := 0;
    Provenance_Continuity_Epoch_Coherent : BOOL := FALSE;

    // Temporal authority.
    Provenance_Continuity_Last_Update_MS : UDINT := 0;
    Provenance_Continuity_Lease_Expired : BOOL := TRUE;

    // Diagnostics.
    Provenance_Continuity_Last_Error_Code : UDINT := 0;
    Provenance_Continuity_Last_Error_Text : STRING(160) := '';
    Provenance_Continuity_Invalidation_Count : UDINT := 0;
END_VAR

(* ---- GVL_RECOVERY_ORDERING_INTEGRITY_FABRIC.gvl ---- *)
VAR_GLOBAL
    Recovery_Ordering_Integrity_Valid : BOOL := FALSE;
    CrossDomain_Recovery_Ordering_Stable : BOOL := FALSE;
    Recovery_Authority_Sequencing_Canonical : BOOL := FALSE;
    Physical_Reactivation_Topology_Safe : BOOL := FALSE;

    Recovery_Ordering_Causality_Valid : BOOL := FALSE;
    Distributed_Recovery_Ordering_Consensus : BOOL := FALSE;

    Unsafe_Recovery_Reordering_Detected : BOOL := FALSE;
    CrossDomain_Reactivation_Race : BOOL := FALSE;
    Recovery_Topology_Divergence : BOOL := FALSE;
    Residual_Unsafe_Reactivation_Detected : BOOL := FALSE;

    Recovery_Ordering_Epoch : UDINT := 0;
END_VAR

(* ---- GVL_RESOURCE_STARVATION_BOUNDARY_FABRIC.gvl ---- *)
VAR_GLOBAL
    Resource_Starvation_Boundary_Valid : BOOL := FALSE;
    Resource_Starvation_Boundary_Granted : BOOL := FALSE;

    Resource_Starvation_Bounded : BOOL := FALSE;
    Fair_Execution_Scheduling_Valid : BOOL := FALSE;
    Distributed_Resource_Allocation_Stable : BOOL := FALSE;

    Resource_Causality_Grounded : BOOL := FALSE;
    Starvation_Recovery_Stable : BOOL := FALSE;

    Resource_Starvation_Detected : BOOL := FALSE;
    Scheduler_Starvation_Detected : BOOL := FALSE;
    Distributed_Allocation_Deadlock_Detected : BOOL := FALSE;

    Resource_Starvation_Epoch : UDINT := 0;
END_VAR

(* ---- GVL_RUNTIME_BUDGET_ENFORCEMENT.gvl ---- *)
VAR_GLOBAL
    // Runtime budget observability.
    Runtime_Budget_Enforcement_Active : BOOL := TRUE;
    Runtime_Budget_Enforcement_ReadOnly : BOOL := TRUE;

    Verification_Runtime_Budget_Observed : BOOL := FALSE;
    Observability_Runtime_Budget_Observed : BOOL := FALSE;
    Diagnostics_Runtime_Budget_Observed : BOOL := FALSE;
    Governance_Runtime_Overhead_Observed : BOOL := FALSE;

    Runtime_Budget_Pressure_Observed : BOOL := FALSE;
    Verification_Time_Budget_Exceeded : BOOL := FALSE;
    Observability_Amplification_Budget_Exceeded : BOOL := FALSE;
    Diagnostics_Load_Budget_Exceeded : BOOL := FALSE;

    Runtime_Stability_Budget_At_Risk : BOOL := FALSE;
    Verification_Induced_Runtime_Risk : BOOL := FALSE;

    Runtime_Budget_Enforcement_Epoch : UDINT := 0;
END_VAR

(* ---- GVL_Runtime_Discovery.gvl ---- *)
{attribute 'qualified_only'}
VAR_GLOBAL RETAIN
    G_Discovery_State : ARRAY[1..32] OF ST_Runtime_Node_Discovery_State;
END_VAR

VAR_GLOBAL
    G_Runtime_Valid : BOOL;
    G_Last_Update_MS : UDINT;

    G_Any_Node_Quarantined : BOOL;
    G_Any_Discovery_Rejected : BOOL;

    G_Status_Code : UINT;
    G_Status_Text : STRING(160);
END_VAR

(* ---- GVL_RUNTIME_RESOURCE_AUTHORITY.gvl ---- *)
VAR_GLOBAL
    // Global runtime resource authority.
    Runtime_Resource_Authority_Valid : BOOL := FALSE;
    Runtime_Resource_Authority_Granted : BOOL := FALSE;
    Runtime_Resource_Quarantine_Active : BOOL := TRUE;

    // Deterministic runtime guarantees.
    Deterministic_Cycle_Time_Valid : BOOL := FALSE;
    Task_Jitter_Within_Bounds : BOOL := FALSE;
    Watchdog_Margin_Stable : BOOL := FALSE;
    Runtime_Latency_Stable : BOOL := FALSE;
    Queue_Backlog_Stable : BOOL := FALSE;

    // Runtime execution metrics.
    Current_Task_Jitter_US : UDINT := 0;
    Max_Allowed_Task_Jitter_US : UDINT := 10000;

    Current_Runtime_Latency_US : UDINT := 0;
    Max_Allowed_Runtime_Latency_US : UDINT := 20000;

    Current_Fieldbus_Queue_Depth : UDINT := 0;
    Max_Allowed_Fieldbus_Queue_Depth : UDINT := 100;

    Current_Watchdog_Margin_MS : UDINT := 0;
    Minimum_Watchdog_Margin_MS : UDINT := 50;

    // Resource exhaustion detection.
    Hidden_Jitter_Amplification_Detected : BOOL := FALSE;
    Queue_Induced_Authority_Lag_Detected : BOOL := FALSE;
    Watchdog_Near_Death_Oscillation_Detected : BOOL := FALSE;
    Runtime_Starvation_Race_Detected : BOOL := FALSE;
    Cycle_Collapse_SplitBrain_Detected : BOOL := FALSE;
    Heap_Fragmentation_Critical : BOOL := FALSE;
    Fieldbus_Backlog_Saturation_Detected : BOOL := FALSE;

    // Runtime authority epochs.
    Runtime_Resource_Authority_Epoch : UDINT := 0;
    Runtime_Resource_Authority_Epoch_Coherent : BOOL := FALSE;

    // Temporal runtime authority.
    Runtime_Resource_Last_Update_MS : UDINT := 0;
    Runtime_Resource_Lease_Expired : BOOL := TRUE;

    // Diagnostics.
    Runtime_Resource_Last_Error_Code : UDINT := 0;
    Runtime_Resource_Last_Error_Text : STRING(160) := '';
    Runtime_Resource_Invalidation_Count : UDINT := 0;
END_VAR

(* ---- GVL_Runtime_Sessions.gvl ---- *)
{attribute 'qualified_only'}
VAR_GLOBAL RETAIN
    G_Local_Session : ST_Runtime_Node_Session;
    G_Remote_Sessions : ARRAY[1..16] OF ST_Runtime_Node_Session;
END_VAR

VAR_GLOBAL
    G_Runtime_Valid : BOOL;
    G_Last_Update_MS : UDINT;

    G_Any_Stale_Session : BOOL;
    G_Any_Quarantined_Session : BOOL;

    G_Status_Code : UINT;
    G_Status_Text : STRING(160);
END_VAR

(* ---- GVL_RUNTIME_SNAPSHOT.gvl ---- *)
VAR_GLOBAL
    // ======================================================
    // IMMUTABLE RUNTIME SNAPSHOT AUTHORITY STATE
    // ======================================================
    // Centralized immutable publication snapshot governance.
    // Prevents mutable publication leakage across cycle boundaries.
    // ======================================================

    Snapshot_Epoch : ULINT := 0;
    Snapshot_Publication_Epoch : ULINT := 0;

    Snapshot_Frozen : BOOL := FALSE;
    Snapshot_Publication_Allowed : BOOL := FALSE;

    Snapshot_Copy_Valid : BOOL := FALSE;
    Snapshot_Isolation_Valid : BOOL := FALSE;
    Snapshot_Mutation_Detected : BOOL := FALSE;

    Snapshot_Runtime_Authority_Valid : BOOL := FALSE;

    Snapshot_Freeze_Start_MS : UDINT := 0;
    Snapshot_Last_Publication_MS : UDINT := 0;

    Snapshot_Last_Error_Code : UDINT := 0;
    Snapshot_Last_Error_Text : STRING(160) := '';
END_VAR

(* ---- GVL_RUNTIME_SUSTAINABILITY_FABRIC.gvl ---- *)
VAR_GLOBAL
    // Global deterministic runtime sustainability authority.
    Runtime_Sustainability_Valid : BOOL := FALSE;
    Runtime_Sustainability_Granted : BOOL := FALSE;
    Runtime_Sustainability_Quarantine_Active : BOOL := TRUE;

    // Sustainable runtime execution proofs.
    Deterministic_Cycle_Budget_Stable : BOOL := FALSE;
    Runtime_Queue_Load_Stable : BOOL := FALSE;
    Memory_Fragmentation_Stable : BOOL := FALSE;
    Watchdog_Jitter_Stable : BOOL := FALSE;
    HA_Synchronization_Load_Stable : BOOL := FALSE;

    // Long-term operational sustainability.
    Historical_Persistence_Load_Stable : BOOL := FALSE;
    Snapshot_Publication_Stable : BOOL := FALSE;
    Distributed_Runtime_Load_Coherent : BOOL := FALSE;
    Runtime_Evolution_Sustainable : BOOL := FALSE;

    // Resource-collapse detectors.
    Memory_Fragmentation_Drift_Detected : BOOL := FALSE;
    Queue_Saturation_Detected : BOOL := FALSE;
    Historical_Persistence_Amplification_Detected : BOOL := FALSE;
    Watchdog_Jitter_Escalation_Detected : BOOL := FALSE;
    HASynchronization_Overload_Detected : BOOL := FALSE;
    Deterministic_Cycle_Erosion_Detected : BOOL := FALSE;

    // Sustainability epochs.
    Runtime_Sustainability_Epoch : UDINT := 0;
    Runtime_Sustainability_Epoch_Coherent : BOOL := FALSE;

    // Temporal authority.
    Runtime_Sustainability_Last_Update_MS : UDINT := 0;
    Runtime_Sustainability_Lease_Expired : BOOL := TRUE;

    // Diagnostics.
    Runtime_Sustainability_Last_Error_Code : UDINT := 0;
    Runtime_Sustainability_Last_Error_Text : STRING(160) := '';
    Runtime_Sustainability_Invalidation_Count : UDINT := 0;
END_VAR

(* ---- GVL_SEMANTIC_FEDERATION_FABRIC.gvl ---- *)
VAR_GLOBAL
    // Global deterministic semantic federation authority.
    Semantic_Federation_Valid : BOOL := FALSE;
    Semantic_Federation_Granted : BOOL := FALSE;
    Semantic_Federation_Quarantine_Active : BOOL := TRUE;

    // External ecosystem semantic coherence proofs.
    External_SCADA_Semantics_Coherent : BOOL := FALSE;
    Cloud_Authority_Projection_Aligned : BOOL := FALSE;
    MQTT_Semantic_State_Fresh : BOOL := FALSE;
    ThirdParty_Integration_Trust_Valid : BOOL := FALSE;
    Federated_Observability_Coherent : BOOL := FALSE;

    // Cross-ecosystem semantic synchronization.
    Exported_Authority_State_Coherent : BOOL := FALSE;
    Federation_Projection_Temporal_Stable : BOOL := FALSE;
    External_Runtime_Interpretation_Aligned : BOOL := FALSE;
    Federated_Trust_Boundary_Stable : BOOL := FALSE;

    // Ecosystem semantic split-brain detectors.
    External_Semantic_Lag_Detected : BOOL := FALSE;
    SCADA_Projection_Skew_Detected : BOOL := FALSE;
    Cloud_Authority_Desynchronization_Detected : BOOL := FALSE;
    ThirdParty_Semantic_Drift_Detected : BOOL := FALSE;
    Integration_Trust_Divergence_Detected : BOOL := FALSE;
    Federated_Authority_Inconsistency_Detected : BOOL := FALSE;

    // Federation epochs.
    Semantic_Federation_Epoch : UDINT := 0;
    Semantic_Federation_Epoch_Coherent : BOOL := FALSE;

    // Temporal authority.
    Semantic_Federation_Last_Update_MS : UDINT := 0;
    Semantic_Federation_Lease_Expired : BOOL := TRUE;

    // Diagnostics.
    Semantic_Federation_Last_Error_Code : UDINT := 0;
    Semantic_Federation_Last_Error_Text : STRING(160) := '';
    Semantic_Federation_Invalidation_Count : UDINT := 0;
END_VAR

(* ---- GVL_SEMANTIC_PRESERVATION_FABRIC.gvl ---- *)
VAR_GLOBAL
    // Global deterministic semantic preservation authority.
    Semantic_Preservation_Valid : BOOL := FALSE;
    Semantic_Preservation_Granted : BOOL := FALSE;
    Semantic_Preservation_Quarantine_Active : BOOL := TRUE;

    // Immutable intent preservation proofs.
    Declared_System_Intent_Coherent : BOOL := FALSE;
    Adaptive_Policy_Bounded : BOOL := FALSE;
    Cross_Domain_Intent_Aligned : BOOL := FALSE;
    Optimization_Goals_Coherent : BOOL := FALSE;
    Behavioral_Evolution_Stable : BOOL := FALSE;

    // Long-term semantic governance coherence.
    Objective_Boundaries_Immutable : BOOL := FALSE;
    Semantic_Governance_Coherent : BOOL := FALSE;
    Adaptive_Runtime_Intent_Stable : BOOL := FALSE;
    LongTerm_Semantic_Evolution_Valid : BOOL := FALSE;

    // Semantic drift detectors.
    Adaptive_Policy_Drift_Detected : BOOL := FALSE;
    Optimization_Semantic_Erosion_Detected : BOOL := FALSE;
    CrossDomain_Intent_Divergence_Detected : BOOL := FALSE;
    LongTerm_Objective_Mutation_Detected : BOOL := FALSE;
    Behavior_Learning_Instability_Detected : BOOL := FALSE;
    Silent_Governance_Reinterpretation_Detected : BOOL := FALSE;

    // Semantic preservation epochs.
    Semantic_Preservation_Epoch : UDINT := 0;
    Semantic_Preservation_Epoch_Coherent : BOOL := FALSE;

    // Temporal authority.
    Semantic_Preservation_Last_Update_MS : UDINT := 0;
    Semantic_Preservation_Lease_Expired : BOOL := TRUE;

    // Diagnostics.
    Semantic_Preservation_Last_Error_Code : UDINT := 0;
    Semantic_Preservation_Last_Error_Text : STRING(160) := '';
    Semantic_Preservation_Invalidation_Count : UDINT := 0;
END_VAR
